DATA_BLOCK "dbdane"   // DB2
{ S7_Optimized_Access := 'FALSE' }
VERSION : 0.1
// stored: AutoNumber true, DBAccessibleFromOPCUA true, IsOnlyStoredInLoadMemory false, IsWriteProtectedInAS false
   VAR RETAIN
      TMR_ON_K3 : Time := T#10s;   // Czas histerezy na dołączenie dodatkowej 3 / Wartość timera na dołączenie drugiej dodatkowej
      amplituda : Real := 95.0;   // Wiekośc zadana amplituda sygnału
      TMR_OFF_K3 : Time := T#10s;   // Czas na odłączenie dodatkowej 3 / Wartość timera na odłączenie drugiej dodatkowej
      Manual_SV : Real;   // Wartość setpint zadana manualnie
      MV : Real;   // Wartość procentowa wyjącia regulatora PID [%]
      PV : Real;   // Wartość liczbowa sygnału analogowego cisnienia tłocznym / Wartość liczbowa sygnału analogowego AI0 bar ciśnienie tłoczenia t
      tuning : Bool;
      zewnetrzne : Bool;
      dzialanie : Bool;
      Setpoint_SV : Real;   // Ciśnienie zadane do regulatora / Wartość zadanego ciśnienia do PID
      WYL : Bool;
      zerowanie : Bool;
      z_obiektu_analog : Word;
      do_obiektu_analog : Word;
      do_obiektu_pwm : Bool;
      PV_PER_B6 : Word;   // Ciśnienie tłoczny miasto (4-20mA) / Ciśnieie Tłoczenia Tłoczny sygnał z wejścia analogowego AI0 bar (4-20mA)
      OUT_PER : Word;   // Sygnał wyjściowy Hz postać procesowa / Sygnał wyjściowy Hz postać analogowa 0-20mA
      TMR_ON_K1 : Time;   // Wartość timera na dołączenie
      TMR_ON_K2 : Time;   // Wartość timera na dołączenie
      TMR_OFF_K1 : Time;   // Wartość timera na odłączenie
      TMR_OFF_K2 : Time;   // Wartość timera na odłączenie
      TMR_Hz : Time;   // Wartość timera na oczykiwanie 50Hz
      HMI : Struct
         PhysicalUnit : String[5] := '1/min';
         Output_PWM_USInt : USInt;
         ManualEnable_edge : Bool;
         ManualMode_visible : Bool;
         "sPid_Cmpt.b_Input_PER_On" : Bool;
         ErrorBits_Int : Int;
         ErrorAck_Int : Int;
         Warning_Int : Int;
         ErrorAck_Int_edge : Bool;
         ErrorAck : Bool;
         Acknowledge_visible : Bool;
         "sPid_Cmpt.r_Pv_Norm_OUT_2" : Real;   // Max wartośc procesowa przekazana z HMI
      END_STRUCT;
      OUT_PURE_Real : Real;   // Sygnał Hz w po scalowaniu do Hz
      Edge_1Hz_P1 : Bool;   // Pamięć zbocza naraztającego dla licznika pracy / Pamięć zbocza naraztającego dla licznika pracy pompy
      Edge_1Hz_P2 : Bool;   // Pamięć zbocza naraztającego dla licznika pracy / Pamięć zbocza naraztającego dla licznika pracy pompy
      Edge_1Hz_P3 : Bool;   // Pamięć zbocza naraztającego dla licznika pracy / Pamięć zbocza naraztającego dla licznika pracy pompy
      Edge_1Hz_P4 : Bool;   // Pamięć zbocza naraztającego dla licznika pracy pompy
      "PID_Compact_1_sPid_Cmpt.r_Lmn_Hlm" : Real;
      "PID_Compact_1sPid_Cmpt.r_Pv_Norm_OUT_2" : Real;
      PID_Compact_1_ManualEnable : Bool;
      PID_Compact_1_ManualValue { ExternalWritable := 'False'} : Real;
      "PID_Compact_1_sPid_Cmpt.r_Lmn_Llm" : Real;
      "PID_Compact_1_sPid_Cmpt.r_Lmn_Pwm_PBTm" : Real;
      "PID_Compact_1_sPid_Cmpt.r_Lmn_Pwm_PPTm" : Real;
      "PID_Compact_1_sPid_Cmpt.r_Pv_HWrn" : Real;   // Nastawa progu ostrzerzenia PV wysoki
      "PID_Compact_1_sPid_Cmpt.r_Pv_LWrn" : Real;   // Nastawa progu ostrzerzenia PV niski
      "PID_Compact_1_sPid_Cmpt.r_Pv_Norm_IN_1" : Real;
      "PID_Compact_1_sPid_Cmpt.r_Pv_Norm_IN_2" : Real;
      "PID_Compact_1_sPid_Cmpt.r_Pv_Norm_OUT_1" : Real;
      "PID_Compact_1_sPid_Cmpt.r_Sp_Hlm" : Real;
      "PID_Compact_1_sPid_Cmpt.r_Sp_Llm" : Real;
      "PID_Compact_1_sPid_Cmpt.r_Pv_Hlm" : Real;
      "PID_Compact_1_sPid_Cmpt.r_Pv_Llm" : Real;
      Setpoint_bar_automat : Real;   // Zadana wartość ciśnienia w trybie automat (sterownik pobiera określoną wartośc zadaną w zależności od kierunku pompowania) / Ciśnienie w magistrali (bobrane ze sterownika Zasuwy) skalowany
      PV_PER_B8 : Word;   // Ciśnienie ssanie suchobieg (4-20mA) / Ciśnienie po stronie ssącej pomp (sychobieg)
      MV_Real_b : Word;
      actPrzepływQ1_Real : Real;   // przepływ pompownia / Aktualny przepływ POMPOWNIA
      actPrzepływQ2_Real : Real;   // Zadane Hz pompomieszadło Word / Aktualny przepływ EC STUDNIA POMIAROWA
      Switch_model_control_Tanks : Word;   // Sygnał sterowania zbiornikami -strategia
      Z11_Status : Word;
      Z12_Status : Word;
      Temp_SV : Word;   // Tymczasowa zadana wartość Hz
      Switch_model_control_P1P4 : Word;   // Sygnały sterowania strategią pompownia - 0= wyłaczone, 1=dosilanie, 2=przetłaczanie,3=automat, 4=ręczne / Model sterowania pompownią (1-dobowe , 2-tygodniowe , 3-Sterowanie standard
      tmp_Hz_ModeAlarm : Real;   // Przechwycone Hz podczas wystąpienia alarmu od max ciśnienie, prąd / Przechwycone Hz podczas wytąpienia alarmu od max ciśnienie, prąd
      actPrzeoływQ1 { ExternalVisible := 'False'} : Int;   // Zmienna aktualny przepływ pompowia / aktualny przepływ Studnia pomiarowa EC Moszczenica
      actPrzepływQ1_IA : Int := 0;   // Zmienna po konwersji do Integer / aktualny przepływ z wejcia analgowego Pompownia jeśli (-) to przepływ wsteczny
      Act_Value_B5_magistrala_bar : Real;   // Zmienna aktualnej wartości ciśnienia magistrala z PLC Zasuwy / Zmienna aktualnej wartości ciśnieniea wspólna Modbus i 4-20mA
      actHz_QW64 : Real := 0.0;   // Zmienna Hz pobrane z wyjacia analogowego / Zmienna aktualnej wartości ciśnieniea wspólna Modbus i 4-20mA
      actPrzepływQ1_IA_real : Real;   // aktualny przepływ Q1 pompownia z wyjścia analogowego / Śerdnia wartość ciśnienie B5 B9
      PV_PER_B7 : Word;   // Ciśnienie tłoczny pompownia(4-20mA) / Ciśnieie Tłoczenia Pompy sygnał z wejścia analogowego AI0 bar (4-20mA)
      act_Value_B6 : Real;   // Ciśnienie tłoczny miasto (Real) / Zmienna aktualnej wartości ciśnieniea B6 po skalowaniau z wejścia (Ciśnieie Tłoczenia Miasto)
      act_Value_B7 : Real;   // Ciśnienie tłoczny pompownia (Real) / Zmienna aktualnej wartości ciśnieniea B7 po skalowaniau z wejścia (Ciśnienie pomp )
      act_Value_B8 : Real;   // Zmienna aktualnej wartości ciśnieniea B5 po skalowaniau z wejścia (Ciśnieie dosilania B5 ) / Ciśnienie ssania (Real)
      tmpdata_MV_PER : Word;   // Tymczasowa aktualnych Hz na potrzeby SCADA przekaznie między tymczasowym Hz a z regulatora PID
      tmpManualSV : LReal;   // pomocnicza przy konwersji wartość zadana manualnie SV
      ManualSV_Int : Int;   // wartość zadana manualnie SV (Word)
      tmpSV_manual_Hold : Int;   // tymczasowa wartość Hz w postaci procesowej podawana na wyjście w czasie podtrzymywania pompy wiodącej po odłaczeniu dodatkowej / tymczasowa wartość Hz w postaci procesowej podawana na wyjście w czasie podtrzymywania dmuchawy wiodącej po odłaczeniu dodatkowej
      tmp_TR_ON_K1_1 : Int := 300;   // Zmienna czasu na dołączenie dodatkowej 1 pobierana przez algorytm PLC
      tmp_TR_ON_K2_1 : Int := 60;   // Zmienna czasu na dołączenie dodatkowej 2 pobierana przez algorytm PLC
      tmp_TR_OFF_K1_1 : Int := 5;   // Zmienna czasu na odołączenie dodatkowej 1 pobierana przez algorytm PLC
      tmp_TR_OFF_K2_1 : Int := 3;   // Zmienna czasu na odołączenie dodatkowej 2 pobierana przez algorytm PLC
      tmp_TR_50Hz_1 : Int := 15;   // Zmienna oczekiwania na 50Hz pobierana przez algorytm PLC
      tmp_TR_ON_K1_2 : Int := 30;   // Zmienna czasu na dołączenie dodatkowej 1 pobierana przez algorytm PLC
      tmp_TR_ON_K2_2 : Int := 30;   // Zmienna czasu na dołączenie dodatkowej 2 pobierana przez algorytm PLC
      tmp_TR_OFF_K1_2 : Int := 5;   // Zmienna czasu na odołączenie dodatkowej 1 pobierana przez algorytm PLC
      tmp_TR_OFF_K2_2 : Int := 5;   // Zmienna czasu na odołączenie dodatkowej 2 pobierana przez algorytm PLC
      tmp_TR_50Hz_2 : Int := 30;   // Zmienna oczekiwania na 50Hz pobierana przez algorytm PLC
      tmp_TR_ON_K1_3 : Int := 5;   // Zmienna czasu na dołączenie dodatkowej 1 pobierana przez algorytm PLC
      tmp_TR_ON_K2_3 : Int := 15;   // Zmienna czasu na dołączenie dodatkowej 2 pobierana przez algorytm PLC
      tmp_TR_OFF_K1_3 : Int := 2;   // Zmienna czasu na odołączenie dodatkowej 1 pobierana przez algorytm PLC
      tmp_TR_OFF_K2_3 : Int := 2;   // Zmienna czasu na odołączenie dodatkowej 2 pobierana przez algorytm PLC
      tmp_TR_50Hz_3 : Int := 5;   // Zmienna oczekiwania na 50Hz pobierana przez algorytm PLC
      tmpSV_spadekBar : Int;   // Hz tymczasowe dla spatku bar Max po odłączeniu dodatkowej / Hz tymczasowe dla opadającego ciśnienia z Max po odłączeniu dodatkowej
      Alarm_Max_bar : Real;   // Alarmowa wartość bar natychmiastowe wyłączenie układu / Alarmowa wartość tlenu natychmiastowe wyłączenie układu
      tmpSV_spadek : Int := 15000;   // pomocnicza Hz tymczasowe dla opadającego ciśnienie z Max / pomocnicza Hz tymczasowe dla opadającego ciśnienia z Max
      addressModbus_Fal : Byte;   // adres modbas urządzenia falownik
      addressModbus_Q1_MPP04 : Byte;   // adres modbas urządzenia przepłuwomierz Q1
      addressModbus_Q2_MPP04 : Byte;   // adres modbas urządzenia przepływomierz Q2
      addressModbus_SlaveID : Byte;   // adres modbas ID slave
      Wielkość_przeływu_Q1 : Real;
      Licznik_objętość_VF_Q1 : Real;
      Licznik_objętość_VR_Q1 : Real;
      Licznik_różnicowy_VD_Q1 : Real;
      Stan_licz_bjętości_GF_Q1 : Real;
      Stan_licz_rózicowego_obj_GD_Q1 : Real;
      _Stan_urządzenia_Q1 : Int;
      Wielkość_przeływu_Q2 : Real;
      Licznik_objętość_VF_Q2 : Real;
      Licznik_objętość_VR_Q2 : Real;
      Licznik_różnicowy_VD_Q2 : Real;
      Stan_licz_bjętości_GF_Q2 : Real;
      Stan_licz_rózicowego_obj_GD_Q2 : Real;
      _Stan_urządzenia_Q2 : Int;
      PV_analaog_B6 : Int;   // wartość analogowa z wejścia AI
      PV_analaog_B7 : Int := 0;   // wartość analogowa z wejścia AI
      PV_analaog_B8 : Int := 0;   // wartość analogowa z wejścia AI
   END_VAR
BEGIN
END_DATA_BLOCK

DATA_BLOCK "dbtags_Sterowanie"   // DB1
{ S7_Optimized_Access := 'FALSE' }
VERSION : 0.1
// stored: AutoNumber false, DBAccessibleFromOPCUA true, IsOnlyStoredInLoadMemory false, IsWriteProtectedInAS false
   VAR RETAIN
      PID_Compact : Struct
         Setpoint : Real := 1.5;
         Input : Real;
         Input_PER : Int;
         Disturbance : Real;
         ManualEnable : Bool;
         ManualValue : Real;
         ErrorAck : Bool;
         Reset : Bool;
         ModeActivate : Bool;
         Mode : Int := 3;
         ScaledInput : Real;
         Output : Real;
         Output_PER : Int;
         Output_PWM : Bool;
         SetpointLimit_H : Bool;
         SetpointLimit_L : Bool;
         InputWarning_H : Bool;
         InputWarning_L : Bool;
         State : Int;
         Error : Bool;
         ErrorBits : DWord;
      END_STRUCT;
      Tuning : Struct
         Mode : Int := 1;
         Mode_visible : Bool;
         SUT_visible : Bool;
         TIR_visible : Bool;
         last_state : Int;
      END_STRUCT;
      HMI : Struct
         PhysicalUnit : String[5] := '1/min';
         Output_PWM_USInt : USInt;
         "position reached" : Bool;
         ManualMode_visible : Bool;
         Setpoint_limited : Bool;
         ErrorBits_Int : Int;
         ErrorAck_Int : Int;
         Warning_Int : Int;
         ErrorAck_Int_edge : Bool;   // pamięć zbocza reset PID po error
         ErrorAck : Bool;   // reset błędu PID
         Acknowledge_visible : Bool;
      END_STRUCT;
      Speed : Struct
         encoder : Real;
         rpm : Real;
      END_STRUCT;
      SetupControlPompownia : Struct
         SV : Real := 2.0;
         r_Pv_Norm_OUT_2 : Real := 10.0;   // Zakres górny wejścia In_PER_PID
         r_Pv_Norm_OUT_1 : Real := 0.0;   // Zakres dolny wejścia In_PER_PID
         r_Lmn_Hlm : Real := 100.0;   // Ograniczenie górne wartości procesowej [%] MV
         r_Lmn_Llm : Real := 0.0;   // Ograniczenie dolne wartości procesowej [%] MV
         r_Sp_Hlm : Real := 10.0;   // Ograniczenie H zakresu zadawania wartości ciśnienie SV
         r_Sp_Llm : Real := 0.0;   // Ograniczenie L zakresu zadawania wartości ciśnienia SV
         r_Pv_HWrn : Real;   // Ostrzeżenie wysoki dla PV
         r_Pv_LWrn : Real;   // Ostrzeżenie niski dla PV
         r_Pv_Hlm : Real := 16.0;   // Przetwornik Limit górny
         r_Pv_Llm : Real := 0.0;   // Przetwornik Limit dlolny
         Time_ONK1 : Int := 20;
         Time_ONK2 : Int := 60;
         Time_OFFK1 : Int := 15;
         Time_OFFK2 : Int := 5;
         TimeHz : Int := 10;
         NO4_Cureent : Real;   // Aktualna zawartość amoniaku
         CureentValue_O2_1 : Real;   // Przyrost ciśnienia 1
         CureentValue_O2_2 : Real;   // Przyrost ciścienia 2
         Data_sek1 : Int;   // Licznik sekund dla pomiaru nr1 funkcji Calculation_of_the_increment
         Data_sek2 : Int;   // Licznik sekund dla pomiaru nr2 funkcji Calculation_of_the_increment
         Static_1 : Word;
         Z11_Status : Word;   // Status napędu copia z SCADA
         Z12_Status : Word;   // Status napędu copia z SCADA
         Static_2 : Real;
         Switch_Aut_Rem_Pompy : Bool;   // Bit przełacznika trybu pracy pomp
         tagsdbSwitch_ModelSterowania : Word;   // Wybur model sterowania0- wyłączone, 1- Dosilanie, 2- Przetłączanie, 3- Automat, 4- Ręczne
         barMax_Manual_Hz : Real := 5.0;   // Instancja wartości zadawanej w trybie manual do regulatora PID gdy ciśnienie w rurociągu max
         CurrentMax_Manual_Hz : Real := 5.0;   // Instancja wartości zadawanej w trybie manual do regulatora PID gdy przeciążony falownik
         Statut_Motor : Byte;   // Byte stanu gotowości pomp
         Mem_Res_setCMD_MC_P1 : Bool;   // Znacznik 50 Hz podtrzymanie przełączenia na sieć
         Mem_Res_setCMD_MC_P2 : Bool;   // Znacznik 50 Hz podtrzymanie przełączenia na sieć
         Mem_Res_setCMD_MC_P3 : Bool;   // Znacznik 50 Hz podtrzymanie przełączenia na sieć
         Switch_In_Analog_Mudbas : Bool;   // Bit przełączeania pomiędzy sygnałem bar z wej analog / Modbus
         PV_HWrn_correction : Real;   // Wspóczninik służący wprowadzeniu korekty ostrzeżenia przekroczenia wartości zadanej ciśnienie
         PV_LWrn_correction : Real;   // Wspóczninik służący wprowadzeniu korekty ostrzeżenia zbyt niskia wartości ciśnieniea w stosunku do zadanej
         TimerSet_O2_Up : IEC_TIMER;   // Czas opóżninia podniesienia zadanej wartości ciśnienia
         TimerSet_O2_Down : IEC_TIMER;   // Czas opóżninia obniżenia zadanej wartości ciśnienia
         Pv_Llm_B8 : Real := -1.0;   // Limit dolny przetwornika ciśnienie B8
         Pv_Hlm_B8 : Real := 2.0;   // Limit górny przetwornika ciśnienia B8
         set_a : Int;
         set_b : Int := 0;
         Setpoint_Inverter_Pompy { ExternalAccessible := 'False'; ExternalVisible := 'False'; ExternalWritable := 'False'} : Real;   // Wartość zadana Hz odczytane z Modbus
         Frequency_inverter_Pompy { ExternalAccessible := 'False'; ExternalVisible := 'False'; ExternalWritable := 'False'} : Real;   // Aktualne Hz silniku odczytane z Modbus
         MotorCurrent_Inverter_Pompy { ExternalAccessible := 'False'; ExternalVisible := 'False'; ExternalWritable := 'False'} : Real;   // Prąd na silniku zasilanym z falownika odczytane z Modbus
         NormalCurrent_InverterPompy { ExternalAccessible := 'False'; ExternalVisible := 'False'; ExternalWritable := 'False'} : Real;   // Prąd nominalny falownika odczytane z Modbus
         MaxCurrent_Inverter_Pompy { ExternalAccessible := 'False'; ExternalVisible := 'False'; ExternalWritable := 'False'} : Real;   // Prad Max krótkotrwały odczytane z Modbus
         OverTemp_InverterPompy { ExternalAccessible := 'False'; ExternalVisible := 'False'; ExternalWritable := 'False'} : Word;
         OverVolta_InverterPompy { ExternalAccessible := 'False'; ExternalVisible := 'False'; ExternalWritable := 'False'} : Word;
         PIF_Reset : IEC_TIMER;   // impuls resetu regulatora PID 1
         mbAdresMPP04_Q1 : Word := 6;   // Adres modbus przepływomierz pompownia
         mbAdresPompy : Word := 26;   // Adres modbus falownik
         mbAdresMPP04_Q2 : Word;   // Adres modbus przepływomierz magistrala - w Stacji Zasuw
         mbAdres_IDslave : Word := 2;   // Adres modbus MT101
         SubPV_K1 : Real := 0.6;   // Wspólczynnik pomniejszenia wyliczanego ciśnienia napotrzeby wyłączenia dodatowej pompy
         SubPV_K2 : Real := 0.45;   // Wspólczynnik pomniejszenia wyliczanego ciśnieia napotrzeby wyłączenia dodatowej pompy
         Setpoint_Inverter_a { ExternalAccessible := 'False'; ExternalVisible := 'False'; ExternalWritable := 'False'} : Real;   // Wartość zadana Hz odczytane z Modbus
         Frequency_inverter_a { ExternalAccessible := 'False'; ExternalVisible := 'False'; ExternalWritable := 'False'} : Real;   // Aktualne Hz silniku odczytane z Modbus
         MotorCurrent_Inverter_a { ExternalAccessible := 'False'; ExternalVisible := 'False'; ExternalWritable := 'False'} : Real;   // Prąd na silniku zasilanym z falownika odczytane z Modbus
         NormalCurrent_Inverter_a { ExternalAccessible := 'False'; ExternalVisible := 'False'; ExternalWritable := 'False'} : Real;   // Prąd nominalny falownika odczytane z Modbus
         MaxCurrent_Inverter_a { ExternalAccessible := 'False'; ExternalVisible := 'False'; ExternalWritable := 'False'} : Real;   // Prad Max krótkotrwały odczytane z Modbus
         OverTemp_InverterPomp { ExternalAccessible := 'False'; ExternalVisible := 'False'; ExternalWritable := 'False'} : Word;
         OverVolta_InverterPomp { ExternalAccessible := 'False'; ExternalVisible := 'False'; ExternalWritable := 'False'} : Word;
         set_barDN500_B5 { ExternalAccessible := 'False'; ExternalVisible := 'False'; ExternalWritable := 'False'} : Real;   // Zadane ciśnienie dosilanie DN500 na czujniku B5
         set_barDN225_B6 { ExternalAccessible := 'False'; ExternalVisible := 'False'; ExternalWritable := 'False'} : Real;   // Zadane ciśnienie przetłacania DN225 na czujniku B6
         MotorCurrent_Inverter_b { ExternalAccessible := 'False'; ExternalVisible := 'False'; ExternalWritable := 'False'} : Real;   // Prąd na silniku zasilanym z falownika odczytane z Modbus
         NormalCurrent_Inverter_b { ExternalAccessible := 'False'; ExternalVisible := 'False'; ExternalWritable := 'False'} : Real;   // Prąd nominalny falownika odczytane z Modbus
         MaxCurrent_Inverter_b { ExternalAccessible := 'False'; ExternalVisible := 'False'; ExternalWritable := 'False'} : Real;   // Prad Max krótkotrwały odczytane z Modbus
         OverTemp_Inverter_b { ExternalAccessible := 'False'; ExternalVisible := 'False'; ExternalWritable := 'False'} : Word;
         OverVolta_Inverter_b { ExternalAccessible := 'False'; ExternalVisible := 'False'; ExternalWritable := 'False'} : Word;
         actOverCurrent_set : Real;   // Zakres ograniczenia prądowego.
         actOverCurrent_set_a : Real := 0.0;   // Zakres ograniczenia prądowego.
         actOverCurrent_set_b : Real := 0.0;   // Zakres ograniczenia prądowego.
         AnalogFrequency_inverter_a { ExternalAccessible := 'False'; ExternalVisible := 'False'; ExternalWritable := 'False'} : Real;   // Aktualne Hz silniku odczytane z Analog
         AnalogFrequency_inverter_b { ExternalAccessible := 'False'; ExternalVisible := 'False'; ExternalWritable := 'False'} : Real := 0.0;   // Aktualne Hz silniku odczytane z Analog
         MaxHour_InverterBlowerWork : Word := 43200;   // Maksymalny czas pracy pracy ciągłej na falowniku dla kompresorów 43200sek = 12h
         TimerSet_Hz_Up_a : IEC_TIMER;
         TimerSet_Hz_Down_a : IEC_TIMER;
         TimerSet_Hz_Up_b : IEC_TIMER;
         TimerSet_Hz_Down_b : IEC_TIMER;
         TimerGen_Hz_Up_a : IEC_TIMER;
         TimerGen_Hz_Down_a : IEC_TIMER;
         TimerGen_Hz_Up_b : IEC_TIMER;
         TimerGen_Hz_Down_b : IEC_TIMER;
         Mem_Res_setCMD_MC_P4 : Bool;   // Znacznik 50 Hz podtrzymanie przełączenia na sieć
         "MPP04_1Master.mode" : Byte := 0;
         "MPP04_2Master.mode" : Byte := 0;
         "Fal_2Master.mode_1" : Byte := 0;
         "Slave_2Master.mode_2" : Byte := 2;
      END_STRUCT;
      "Paramaetry _Zbiorniki" : Struct   // parametry sterowania
         set_poziom_napełniania : Real := 550.0;   // wartość zadana poziomu napełniania
         set_poziom_opróżniania : Real := 30.0;   // wartość zadana poziomu opróżniania
         set_bity_sterowania_napęami_1 : Word;   // bity sterowania napędami
         set_bity_sterowania_napęami_2 : Word;   // bity sterowania napędami
         set_bity_tryb_napędów_1 : Word;   // bity sterowania przełączaniem trybów pracy
         set_bity_tryb_napędów_2 : Word;   // bity sterowania przełączaniem trybów pracy
         rez_alarm_napędów : Word;   // bity kasowania alarmów napędów
         set_strategia_sterowania : Word;   // Sygnały sterowania strategią pompownia - 0= wyłaczone, 1=dosilanie, 2=przetłaczanie,3=automat, 4=ręczne
         set_sterowanie_cyklem : Word;   // Sygnały sterowania cyklem zbiorniki 0-wyłączone, 1=dobowy, 2=tygodniowy, 3=ręczne
         set_położenie_Z10 : Word;   // zadane położenie procentowe Z10
      END_STRUCT;
      Zbiorniki_Godziny : Struct   // godziny cykli pracy
         start_napełnianie : DTL := DTL#1970-01-01-23:55:00;
         Stop_napełnianie : DTL := DTL#1970-01-01-16:00:00;
         Start_przetłaczanie_1 : DTL := DTL#1970-01-01-18:00:00;
         Stop_przetłaczanie_1 : DTL := DTL#1970-01-01-23:55:00;
         Start_dosilanie_1 : DTL := DTL#1970-01-01-18:00:00;
         Stop_dosilanie_1 : DTL := DTL#1970-01-01-23:55:00;
      END_STRUCT;
   END_VAR
BEGIN
   SetupControlPompownia.PIF_Reset.PT := T#500ms;
   SetupControlPompownia.TimerSet_Hz_Up_a.PT := T#2M;
   SetupControlPompownia.TimerSet_Hz_Down_a.PT := T#2M;
   SetupControlPompownia.TimerSet_Hz_Up_b.PT := T#2M;
   SetupControlPompownia.TimerSet_Hz_Down_b.PT := T#2M;
   SetupControlPompownia.TimerGen_Hz_Up_a.PT := T#100ms;
   SetupControlPompownia.TimerGen_Hz_Down_a.PT := T#100ms;
   SetupControlPompownia.TimerGen_Hz_Up_b.PT := T#100ms;
   SetupControlPompownia.TimerGen_Hz_Down_b.PT := T#100ms;
END_DATA_BLOCK

DATA_BLOCK "dbMasterData"   // DB35
{ S7_Optimized_Access := 'FALSE' }
VERSION : 0.1
// stored: AutoNumber false, DBAccessibleFromOPCUA true, IsOnlyStoredInLoadMemory false, IsWriteProtectedInAS false
   VAR
      data5_Wielkość_przeływu_Adres_0 { S7_SetPoint := 'True'} : "typeDataMPP04_Int";   // wielkość przepływu / Wartość aktualnego przepływu
      data5_Licznik_objętość_VF_Adres_2 : "typeDataMPP04_Int";   // licznik objętości VF / Stan licznika objętości dla przepływu w przód VF
      data5_Licznik_objętość_VR_Adres_4 { S7_SetPoint := 'True'} : "typeDataMPP04_Int";   // licznik objętości VR / Stan licznika objętości dla przepływu w tył VR
      data5_Licznik_różnicowy_VD_Adres_6 { S7_SetPoint := 'True'} : "typeDataMPP04_Int";   // licznik różnicy / Stan bieżącego różnicowego licznika objętości VD
      data5_Stan_licz_bjętości_GF_Adres_8 { S7_SetPoint := 'True'} : "typeDataMPP04_Int";   // licznik objetosci GF / Stan głównego licznika objętości dla przepływu w przód GF
      data5_Stan_licz_bjętości_GR_Adres_10 { S7_SetPoint := 'True'} : "typeDataMPP04_Int";   // licznik objetości GR / Sta ngłownego licznika objętości dla przepływu w tył GR
      data5_Stan_licz_rózicowego_obj_GD_Adres_12 { S7_SetPoint := 'True'} : "typeDataMPP04_Int";   // licznik róznicowy / Stan głownego licznika różnicowego GD
      data5_Stan_urządzenia_1000 { S7_SetPoint := 'True'} : "typeDataInverter_Word";   // stan urządzenia / 8-przekrodzony zakres pracy przetwornika, 20-otwarty obwód cewki, 21zwarcie w obwodzie cewki, 26-brak cieczy w czujniku
      data6_Wielkość_przeływu_Adres_0 { S7_SetPoint := 'True'} : "typeDataMPP04_Int";   // wielkość przepływu / Wartość aktualnego przepływu
      data6_Licznik_objętość_VF_Adres_2 { S7_SetPoint := 'True'} : "typeDataMPP04_Int";   // licznik objętości VF / Stan licznika objętości dla przepływu w przód VF
      data6_Licznik_objętość_VR_Adres_4 { S7_SetPoint := 'True'} : "typeDataMPP04_Int";   // licznik objętości VR / Stan licznika objętości dla przepływu w tył VR
      data6_Licznik_różnicowy_VD_Adres_6 { S7_SetPoint := 'True'} : "typeDataMPP04_Int";   // licznik różnicy / Stan bieżącego różnicowego licznika objętości VD
      data6_Stan_licz_bjętości_GF_Adres_8 { S7_SetPoint := 'True'} : "typeDataMPP04_Int";   // licznik objetosci GF / Stan głównego licznika objętości dla przepływu w przód GF
      data6_Stan_licz_bjętości_GR_Adres_10 { S7_SetPoint := 'True'} : "typeDataMPP04_Int";   // licznik objetości GR / Sta ngłownego licznika objętości dla przepływu w tył GR
      data6_Stan_licz_rózicowego_obj_GD_Adres_12 { S7_SetPoint := 'True'} : "typeDataMPP04_Int";   // licznik róznicowy / Stan głownego licznika różnicowego GD
      data6_Stan_urządzenia_1000 { S7_SetPoint := 'True'} : "typeDataInverter_Word";   // stan urządzenia / 8-przekrodzony zakres pracy przetwornika, 20-otwarty obwód cewki, 21zwarcie w obwodzie cewki, 26-brak cieczy w czujniku
      data26_Inver_Control_word_416000_Fal { S7_SetPoint := 'True'} : "typeDataInverter_Word";   // Sowo komtrolneCTW falownika [Uint16, index 0]
      data26_Inver_setpoint_ref_416020_Fal { S7_SetPoint := 'True'} : "typeDataInverter_Word";   // Słowo wartość zadana Hz [Int16, index -1]
      data26_Inver_Status_word_416030_Fal { S7_SetPoint := 'True'} : "typeDataInverter_Word";   // Słowo statusu STW falownika [Uint16, index 0]
      data26_Inver_Frequency_416130_Fal { S7_SetPoint := 'True'} : "typeDataInverter_Word";   // Słowo częstotliwość na wyjściu [Uint16, index -1]
      data26_Inver_MotorCurrent_416140_Fal { S7_SetPoint := 'True'} : "typeDataInverter_Word";   // Słowo częstotliwość na wyjściu [Uint16, index -2]
      data26_Inver_DC_Voltage_416300_Fal { S7_SetPoint := 'True'} : "typeDataInverter_Word";   // Słowo napięcia DC na szynie [Uint16, index 0]
      data26_Inver_Temp_416340_Fal { S7_SetPoint := 'True'} : "typeDataInverter_Word";   // Słowo temperatura invertera [Uint8, index 0]
      data26_Inver_NomCurrent_416360_Fal { S7_SetPoint := 'True'} : "typeDataInverter_Word";   // Słowo nominalna wartośc prądu falonika[Uint16, index -2]
      data26_Inver_MaxCurrent_416370_Fal { S7_SetPoint := 'True'} : "typeDataInverter_Word";   // Słowo max prąd falownika [Uint16, index -2]
      data26_Inver_InDigit_416600_Fal { S7_SetPoint := 'True'} : "typeDataInverter_Word";   // Słowo mampa wejść 18,19,27,33 [Uint16, index -0]
      data26_Inver_HourWork_415010_Fal { S7_SetPoint := 'True'} : "typeDataInverter_DWord";   // Podwójne słowo czasu pracy falownika [Int32, index -0]
      data26_Inver_OverTemp_415040_Fal { S7_SetPoint := 'True'} : "typeDataInverter_Word";   // Sowo statusu przekroczenie temperatury[Uint16, index 0]
      data26_Inver_OverVolts_415050_Fal { S7_SetPoint := 'True'} : "typeDataInverter_Word";   // Sowo statusu przekroczenie napięcia[Uint16, index 0]
      data_RTU_value_0 { S7_SetPoint := 'True'} : "typeDataMPP04_real";   // Wartość 0.0 pomocnicza wyświetlana podczas błędu pomiaru
   END_VAR
BEGIN
   data_RTU_value_0.data[0] := 0.0;
END_DATA_BLOCK

DATA_BLOCK "dbModbusRTU_Reg"   // DB37
TITLE = Modbus RTU Data
{ S7_Optimized_Access := 'FALSE' }
AUTHOR : RTecmer
VERSION : 0.1
// Dane pomiarowe przekazane z bloku danych master modbus RTU
// stored: AutoNumber true, DBAccessibleFromOPCUA true, IsOnlyStoredInLoadMemory false, IsWriteProtectedInAS false
   VAR
      received_5_Wielkość_przeływu_Adres_0 { S7_SetPoint := 'True'} : "typeDataMPP04_Int";   // wielkość przepływu
      received_5_Licznik_objętość_VF_Adres_2 { S7_SetPoint := 'True'} : "typeDataMPP04_Int";   // licznik objętości VF
      received_5_Licznik_objętość_VR_Adres_4 { S7_SetPoint := 'True'} : "typeDataMPP04_Int";   // licznik objętości VR
      received_5_Licznik_różnicowy_VD_Adres_6 { S7_SetPoint := 'True'} : "typeDataMPP04_Int";   // licznik różnicy
      receive_5_Stan_licz_bjętości_GF_Adres_8 { S7_SetPoint := 'True'} : "typeDataMPP04_Int";   // licznik objetosci GF
      received_5_Stan_licz_bjętości_GR_Adres_10 { S7_SetPoint := 'True'} : "typeDataMPP04_Int";   // licznik objetości GR
      received_5_Stan_licz_rózicowego_obj_GD_Adres_12 { S7_SetPoint := 'True'} : "typeDataMPP04_Int";   // licznik róznicowy
      received_5_Stan_urządzenia_1000 { S7_SetPoint := 'True'} : "typeDataInverter_Word";   // stan urządzenia
      received_6_Wielkość_przeływu_Adres_0 { S7_SetPoint := 'True'} : "typeDataMPP04_Int";   // wielkość przepływu
      received_6_Licznik_objętość_VF_Adres_2 { S7_SetPoint := 'True'} : "typeDataMPP04_Int";   // licznik objętości VF
      received_6_Licznik_objętość_VR_Adres_4 { S7_SetPoint := 'True'} : "typeDataMPP04_Int";   // licznik objętości VR
      received_6_Licznik_różnicowy_VD_Adres_6 { S7_SetPoint := 'True'} : "typeDataMPP04_Int";   // licznik różnicy
      receive_6_Stan_licz_bjętości_GF_Adres_8 { S7_SetPoint := 'True'} : "typeDataMPP04_Int";   // licznik objetosci GF
      received_6_Stan_licz_bjętości_GR_Adres_10 { S7_SetPoint := 'True'} : "typeDataMPP04_Int";   // licznik objetości GR
      received_6_Stan_licz_rózicowego_obj_GD_Adres_12 { S7_SetPoint := 'True'} : "typeDataMPP04_Int";   // licznik róznicowy
      received_6_Stan_urządzenia_1000 { S7_SetPoint := 'True'} : "typeDataInverter_Word";   // stan urządzenia
      receivede26_Inver_Control_word_416000 { S7_SetPoint := 'True'} : "typeDataInverter_Word";   // Sowo komtrolneCTW falownika [Uint16, index 0]
      received26_Inver_setpoint_ref_416020 { S7_SetPoint := 'True'} : "typeDataInverter_Word";   // Słowo wartość zadana Hz [Int16, index -1]
      received26_Inver_Status_word_416030 { S7_SetPoint := 'True'} : "typeDataInverter_Word";   // Słowo statusu STW falownika [Uint16, index 0]
      received26_Inver_Frequency_416130 { S7_SetPoint := 'True'} : "typeDataInverter_Word";   // Słowo częstotliwość na wyjściu [Uint16, index -1]
      received26_Inver_MotorCurrent_416140 { S7_SetPoint := 'True'} : "typeDataInverter_Word";   // Słowo częstotliwość na wyjściu [Uint16, index -2]
      received26_Inver_DC_Voltage_416300 { S7_SetPoint := 'True'} : "typeDataInverter_Word";   // Słowo napięcia DC na szynie [Uint16, index 0]
      received26_Inver_Temp_416340 { S7_SetPoint := 'True'} : "typeDataInverter_Word";   // Słowo temperatura invertera [Uint8, index 0]
      received26_Inver_NomCurrent_416360 { S7_SetPoint := 'True'} : "typeDataInverter_Word";   // Słowo nominalna wartośc prądu falonika[Uint16, index -2]
      received26_Inver_MaxCurrent_416370 { S7_SetPoint := 'True'} : "typeDataInverter_Word";   // Słowo max prąd falownika [Uint16, index -2]
      received26_Inver_InDigit_416600 { S7_SetPoint := 'True'} : "typeDataInverter_Word";   // Słowo mampa wejść 18,19,27,33 [Uint16, index -0]
      received26_Inver_HourWork_415010 { S7_SetPoint := 'True'} : "typeDataInverter_DWord";   // Podwójne słowo czasu pracy falownika [Int32, index -0]
      received26_Inver_OverTemp_415040 { S7_SetPoint := 'True'} : "typeDataInverter_Word";   // Sowo statusu przekroczenie temperatury[Uint16, index 0]
      received26_Inver_OverVolts_415050 { S7_SetPoint := 'True'} : "typeDataInverter_Word";   // Sowo statusu przekroczenie napięcia[Uint16, index 0]
      "Przepływomierz nr1 pompownia" : Struct
         received_5_przeływu_VF_Adres_0 { S7_SetPoint := 'True'} : Real;
         received_5_objętość_VF_Adres_2 { S7_SetPoint := 'True'} : Real;
         "received_5_objętośc RF_Adres_4" { S7_SetPoint := 'True'} : Real;
         received_5_licznik_różnicowy_VD_Adres_6 { S7_SetPoint := 'True'} : Real;
         received_5_licznik_objętości_GF_Adres_8 { S7_SetPoint := 'True'} : Real;
         received_5_Licznik_objętości_GR_Adres_10 { S7_SetPoint := 'True'} : Real;
         received_5_Licznik_różnicowy_GD_Adres_12 { S7_SetPoint := 'True'} : Real;
         received_5_status_przepływomierza_Adres_1000 { S7_SetPoint := 'True'} : Word;
      END_STRUCT;
      "Przepływomierz nr2 Zasuwy" : Struct
         received_6_przeływu_VF_Adres_0 { S7_SetPoint := 'True'} : Real;
         received_6_objętość_VF_Adres_2 { S7_SetPoint := 'True'} : Real;
         "received_6_objętośc RF_Adres_4" { S7_SetPoint := 'True'} : Real;
         received_6_licznik_różnicowy_VD_Adres_7 { S7_SetPoint := 'True'} : Real;
         received_6_licznik_objętości_GF_Adres_8 { S7_SetPoint := 'True'} : Real;
         received_6_Licznik_objętości_GR_Adres_10 { S7_SetPoint := 'True'} : Real;
         received_6_Licznik_różnicowy_GD_Adres_12 { S7_SetPoint := 'True'} : Real;
         received_6_status_przepływomierza_Adres_1000 { S7_SetPoint := 'True'} : Word;
      END_STRUCT;
   END_VAR
BEGIN
END_DATA_BLOCK

DATA_BLOCK "dbTags_master_Fal_1"   // DB74
{ S7_Optimized_Access := 'FALSE' }
VERSION : 0.1
// stored: AutoNumber true, DBAccessibleFromOPCUA true, IsOnlyStoredInLoadMemory false, IsWriteProtectedInAS false
   VAR
      "step" : USInt := 1;
      edge : Bool := false;
      modbusCommLoad { S7_SetPoint := 'True'} : "typeModbusCommLoad";
      modbusMaster { S7_SetPoint := 'True'} : "typeModbusMaster";
   END_VAR
BEGIN
END_DATA_BLOCK

DATA_BLOCK "dbTags_master_MPP04_1"   // DB38
{ S7_Optimized_Access := 'FALSE' }
VERSION : 0.1
// stored: AutoNumber true, DBAccessibleFromOPCUA true, IsOnlyStoredInLoadMemory false, IsWriteProtectedInAS false
   VAR
      "step" : USInt := 1;
      edge : Bool := false;
      modbusCommLoad { S7_SetPoint := 'True'} : "typeModbusCommLoad";
      modbusMaster { S7_SetPoint := 'True'} : "typeModbusMaster";
   END_VAR
BEGIN
END_DATA_BLOCK

DATA_BLOCK "dbTags_master_MPP04_2"   // DB81
{ S7_Optimized_Access := 'FALSE' }
VERSION : 0.1
// stored: AutoNumber true, DBAccessibleFromOPCUA true, IsOnlyStoredInLoadMemory false, IsWriteProtectedInAS false
   VAR
      "step" : USInt := 1;
      edge : Bool := false;
      modbusCommLoad { S7_SetPoint := 'True'} : "typeModbusCommLoad";
      modbusMaster { S7_SetPoint := 'True'} : "typeModbusMaster";
   END_VAR
BEGIN
END_DATA_BLOCK

DATA_BLOCK "dbTags_master_RTU"   // DB90
TITLE = Master
{ S7_Optimized_Access := 'FALSE' }
AUTHOR : rtecmer
VERSION : 0.1
// Instancja dla funkcji Mdbus RTU komunikacja z masterem MT101
// stored: AutoNumber false, DBAccessibleFromOPCUA true, IsOnlyStoredInLoadMemory false, IsWriteProtectedInAS false
   VAR
      "step" : USInt := 1;
      edge : Bool := false;
      modbusCommLoad { S7_SetPoint := 'True'} : "typeModbusCommLoad";
      modbusMaster { S7_SetPoint := 'True'} : "typeModbusSlave";
   END_VAR
BEGIN
END_DATA_BLOCK

DATA_BLOCK "dbTags_slave_RTU"   // DB79
TITLE = Master
{ S7_Optimized_Access := 'FALSE' }
AUTHOR : rtecmer
VERSION : 0.1
// Instancja dla funkcji Mdbus RTU komunikacja z masterem MT101
// stored: AutoNumber false, DBAccessibleFromOPCUA true, IsOnlyStoredInLoadMemory false, IsWriteProtectedInAS false
   VAR
      "step" : USInt := 1;
      edge : Bool := false;
      modbusCommLoad { S7_SetPoint := 'True'} : "typeModbusCommLoad";
      modbusMaster { S7_SetPoint := 'True'} : "typeModbusSlave";
   END_VAR
BEGIN
END_DATA_BLOCK

DATA_BLOCK "temp_dbHoldRegSlave_to_MT101"   // DB102
{ S7_Optimized_Access := 'FALSE' }
VERSION : 0.1
// stored: AutoNumber false, DBAccessibleFromOPCUA true, IsOnlyStoredInLoadMemory false, IsWriteProtectedInAS false
   VAR
      Status_Sterowanie : Struct
         instPump1 : Int;   // Pompa Status M1
         instPump2 : Int := 0;   // Pompa Status M2
         instPump3 : Int := 0;   // Pompa Status M3
         instPump4 : Int := 0;   // Pompa Status M4
         instvValveZ1 : Int := 0;   // Zasuwa Status Z1
         instvValveZ2 : Int := 0;   // Zasuwa Status Z2
         instvValveZ3 : Int := 0;   // Zasuwa Status Z3
         instvValveZ4 : Int := 0;   // Zasuwa Status Z4
         instvValveZ5 : Int := 0;   // Zasuwa Status Z5
         instvValveZ6 : Int := 0;   // Zasuwa Status Z6
         instvValveZ7 : Int := 0;   // Zasuwa Status Z7
         instvValveZ8 : Int := 0;   // Zasuwa Status Z8
         instvValveZ9 : Int := 0;   // Zasuwa Status Z9
         instvValveZ10 : Int := 0;   // Zasuwa Status Z10
         instvValveZ11 : Int := 0;   // Zasuwa Status Z11
         instvValveZ12 : Int := 0;   // Zasuwa Status Z12
         instControllDrivers_1 : Int := 0;   // Bity sterowania napędami (start, stop, otwórz, zamknij) / Bity sterowania napędami (start, stop, otwórz, zamknij) Pompami M1-M4, Zasuwami Z1, Z2, Z3, Z4
         instControllDrivers_2 : Int := 0;   // Bity przełączenia trybu pracy napędów / Bity sterowania napędami ( otwórz, zamknij, start, stop) Zasuwami Z5, Z6, Z7, Z8, Z9, Z10, Z11, Z12
         instConrol_ManAut_1 : Int := 0;   // Bity przełączenia trybu pracy napędów / Bity przełączenia trybu pracy napędów M1-M4, Zasuwami Z1, Z2, Z3, Z4
         instConrol_ManAut_2 : Int := 0;   // Bity przełączenia trybu pracy napędów / Bity przełączenia trybu pracy napędów Z5, Z6, Z7, Z8, Z9, Z10, Z11, Z12
         instLevelTank1 : Int := 0;   // Poziom zbiornik
         instLevelTank2 : Int := 0;   // Poziom zbiornik
         instLevelTank3 : Int := 0;   // Poziom zbiornik
         instLevelTank4 : Int := 0;   // Poziom zbiornik
         instPosition_Z10 : Int := 0;   // rezerwa / Zadawanie położenia Z10
         instControlClearFault1 : Int := 0;   // Bity kasowania alarmów napędów M1-M4, Z1 - Z12
         instControlSygSter_1 : Int := 0;   // rezerwa / Sygnały sterowania strategią (Bit 53.0 - Wyłączony), (Bit 53.1 - Dosilanie), (Bit 53.2 - Przetłączanie), (Bit 53.3 - Automat), (Bit 53.4 - Ręczne )
         instControlSygSter_2 : Int := 0;   // Sygnały sterowania cyklem (Bit 55.0 - Cykl wyłączony (Bit 55.1 - Cykl dobowy), (Bit 55.2 - Cykl tygodniowy), (Bit 55.3 - Cykl ręczny)
         instCurrent_Inverter : Int := 0;   // Aktualny prądu falownika
         instHz_Inverter : Int := 0;   // Aktualne Hz na falowniku
      END_STRUCT;
      Pomiary : Struct
         instLevelSetfilling : Real;   // Zadany poziom napełniania
         instLevelSetemptying : Real;   // Zadany poziom opróżniania
         instSetbarDN500_B6 : Real;   // Zadany ciśnienie tłóczenia kierunek miasto, Modbus 40035
         instSetbarDN500_B5 : Real;   // Zadana ciśnienie dosilania kierunek dosilanie "0" Modbus 40037
         instSetBarMinB9 : Real;   // Zadawana dolna granica ciśnienia studnia "Granica" Modbus 40039
         instB5bar_act : Real;   // Aktualne ciśnienie zasilania z sieci
         instB6bar_act : Real;   // Aktualne ciśnienie DN225 tłoczny
         instB7bar_act : Real;   // Aktualne ciśnienie DN225 pompy
         instB8bar_act : Real;   // Aktualne ciśnienie ssoncy pomp (zab. Suchobieg)
         instPozitionZ10_act : Real;   // Aktualna pozycja zasuwy Z10
         instFlowDN225_act : Real;   // Przepływ DN225 aktualny MIASTO
         instFlowDN225_sum : Real;   // SUMA przepływu Dolna DN225
         instFlowDN500_act : Real;   // Przepływ DN500 (l/s) aktualny, zasilanie zbiorników, DOSILANIE, Modbus 40055
         instFlowDN500_sum : Real;   // SUMA przepływu Dolna DN500 Modbus 40057
      END_STRUCT;
      Godziny : Struct
         instHourStart_Filling : Int;   // Godzina start napełniania
         instMinutStart_Filling : Int;   // Minuta start napełniania
         instHourStop_Filling : Int;   // Godzina stop napełniania
         instMinutStopt_Filling : Int;   // Minuta stop napełniania
         instHourStart_City : Int;   // Godzina start przetłaczanie miasto DN225
         instMinutStart_City : Int;   // Minuty start przetłaczanie miasto DN225
         instHourStop_City : Int;   // Godzina stop przetłaczanie miasto DN225
         instMinutStopt_City : Int;   // Minuty stop przetłaczanie miasto DN225
         instHourStart_Replen : Int;   // Godzina start przetłaczanie miasto DN225
         instMinutStart_Replen : Int;   // Minuty start przetłaczanie miasto DN225
         instHourStop_Replen : Int;   // Godzina stop przetłaczanie miasto DN225
         instMinutStopt_Replen : Int;   // Minuty stop przetłaczanie miasto DN225
      END_STRUCT;
   END_VAR
BEGIN
END_DATA_BLOCK

DATA_BLOCK "CONFIG_MODBUS_TCP_SERVER"   // DB86
TITLE = CONECT MODBUS TCP SERVER
{ S7_Optimized_Access := 'TRUE' }
AUTHOR : rtecmer
VERSION : 0.1
// stored: AutoNumber true, DBAccessibleFromOPCUA true, IsOnlyStoredInLoadMemory false, IsRetainMemResEnabled false, IsWriteProtectedInAS false, MemoryReserve 100
   VAR
      CONNECT_MODBUS_TCP_Serwer_1 { S7_SetPoint := 'True'} : TCON_IP_v4;
      ERROR_STATUS_SERWER_1 : Word;   // wartość błędu
      ERROR_STATUS_SERWER_2 : Word := 16#0;   // wartość błędu
      ERROR_STATUS_SERWER_3 : Word := 16#0;   // wartość błędu
      ERROR_STATUS_SERWER_4 : Word := 16#0;   // wartość błędu
      "CONFIG SERWER_1" : Struct
         STATUS { S7_SetPoint := 'True'} : Word;   // Status połączenia TCP Modbus
         error : Bool;   // błąd
         dr : Bool;   // dane czytane
         ndr : Bool;   // dane gotowe
      END_STRUCT;
      "CONFIG SERWER_2" : Struct
         STATUS { S7_SetPoint := 'True'} : Word;   // Status połączenia TCP Modbus
         error : Bool;   // błąd
         dr : Bool;   // dane czytane
         ndr : Bool;   // dane gotowe
      END_STRUCT;
      "CONFIG SERWER_3" : Struct
         STATUS { S7_SetPoint := 'True'} : Word;   // Status połączenia TCP Modbus
         error : Bool;   // błąd
         dr : Bool;   // dane czytane
         ndr : Bool;   // dane gotowe
      END_STRUCT;
      "CONFIG SERWER_4" : Struct
         STATUS { S7_SetPoint := 'True'} : Word;   // Status połączenia TCP Modbus
         error : Bool;   // błąd
         dr : Bool;   // dane czytane
         ndr : Bool;   // dane gotowe
      END_STRUCT;
      "CONFIG SERWER_5" : Struct
         STATUS { S7_SetPoint := 'True'} : Word;   // Status połączenia TCP Modbus
         error : Bool;   // błąd
         dr : Bool;   // dane czytane
         ndr : Bool;   // dane gotowe
      END_STRUCT;
      "CONFIG SERWER_6" : Struct
         STATUS { S7_SetPoint := 'True'} : Word;   // Status połączenia TCP Modbus
         error : Bool;   // błąd
         dr : Bool;   // dane czytane
         ndr : Bool;   // dane gotowe
      END_STRUCT;
      "CONFIG SERWER_7" : Struct
         STATUS { S7_SetPoint := 'True'} : Word;   // Status połączenia TCP Modbus
         error : Bool;   // błąd
         dr : Bool;   // dane czytane
         ndr : Bool;   // dane gotowe
      END_STRUCT;
      "CONFIG SERWER_8" : Struct
         STATUS { S7_SetPoint := 'True'} : Word;   // Status połączenia TCP Modbus
         error : Bool;   // błąd
         dr : Bool;   // dane czytane
         ndr : Bool;   // dane gotowe
      END_STRUCT;
      ERROR_STATUS_SERWER_5 : Word := 16#0;   // wartość błędu
      ERROR_STATUS_SERWER_6 : Word := 16#0;   // wartość błędu
      ERROR_STATUS_SERWER_7 : Word := 16#0;   // wartość błędu
      ERROR_STATUS_SERWER_8 : Word := 16#0;   // wartość błędu
   END_VAR
BEGIN
   CONNECT_MODBUS_TCP_Serwer_1.InterfaceId := 64;
   CONNECT_MODBUS_TCP_Serwer_1.ID := 1;
   CONNECT_MODBUS_TCP_Serwer_1.ConnectionType := 11;
   CONNECT_MODBUS_TCP_Serwer_1.LocalPort := 502;
END_DATA_BLOCK

DATA_BLOCK "dbHoldTempMT101"   // DB116
{ S7_Optimized_Access := 'FALSE' }
VERSION : 0.1
// stored: AutoNumber false, DBAccessibleFromOPCUA true, IsOnlyStoredInLoadMemory false, IsWriteProtectedInAS false
   VAR
      Status_Sterowanie : Struct
         instPump1 : Word := 33924;   // Pompa Status M1
         instPump2 : Word := 33924;   // Pompa Status M2
         instPump3 : Word := 33924;   // Pompa Status M3
         instPump4 : Word := 33924;   // Pompa Status M4
         instvValveZ1 : Word := 33924;   // Zasuwa Status Z1
         instvValveZ2 : Word := 33924;   // Zasuwa Status Z2
         instvValveZ3 : Word := 33924;   // Zasuwa Status Z3
         instvValveZ4 : Word := 33924;   // Zasuwa Status Z4
         instvValveZ5 : Word := 33924;   // Zasuwa Status Z5
         instvValveZ6 : Word := 33924;   // Zasuwa Status Z6
         instvValveZ7 : Word := 33924;   // Zasuwa Status Z7
         instvValveZ8 : Word := 33924;   // Zasuwa Status Z8
         instvValveZ9 : Word := 33924;   // Zasuwa Status Z9
         instvValveZ10 : Word := 33924;   // Zasuwa Status Z10
         instvValveZ11 : Word := 33924;   // Zasuwa Status Z11
         instvValveZ12 : Word := 33924;   // Zasuwa Status Z12
         instControllDrivers_1 : Int := 0;   // Bity sterowania napędami (start, stop, otwórz, zamknij) / Bity sterowania napędami (start, stop, otwórz, zamknij) Pompami M1-M4, Zasuwami Z1, Z2, Z3, Z4
         instControllDrivers_2 : Int := 0;   // Bity przełączenia trybu pracy napędów / Bity sterowania napędami ( otwórz, zamknij, start, stop) Zasuwami Z5, Z6, Z7, Z8, Z9, Z10, Z11, Z12
         instConrol_ManAut_1 : Int := 0;   // Bity przełączenia trybu pracy napędów / Bity przełączenia trybu pracy napędów M1-M4, Zasuwami Z1, Z2, Z3, Z4
         instConrol_ManAut_2 : Int := 0;   // Bity przełączenia trybu pracy napędów / Bity przełączenia trybu pracy napędów Z5, Z6, Z7, Z8, Z9, Z10, Z11, Z12
         instLevelTank1 : Int := 0;   // Poziom zbiornik
         instLevelTank2 : Int := 0;   // Poziom zbiornik
         instLevelTank3 : Int := 0;   // Poziom zbiornik
         instLevelTank4 : Int := 0;   // Poziom zbiornik
         instPosition_Z10 : Real := 0.0;   // rezerwa / Zadawanie położenia Z10
         instClearFault1 : Int := 0;   // Bity kasowania alarmów napędów M1-M4, Z1 - Z12
         instSygSter_1 : Int := 2;   // rezerwa / Sygnały sterowania strategią pompownia - 0= wyłaczone, 1=dosilanie, 2=przetłaczanie,3=automat, 4=ręczne
         instSygSter_2 : Int := 1;   // Sygnały sterowania cyklem zbiorniki 0-wyłączone, 1=dobowy, 2=tygodniowy, 3=ręczne
         instCurrent_Inverter : Int := 0;   // Aktualny prądu falownika
         instHz_Inverter : Int := 0;   // Aktualne Hz na falowniku
      END_STRUCT;
      Pomiary : Struct
         instLevelSetFilling : Real := 550.0;   // Zadany poziom napełniania
         instLevelSetEmptying : Real := 10.0;   // Zadany poziom opróżniania
         instSetbarDN225_B6 : Real := 6.6;   // Zadany ciśnienie tłóczenia kierunek miasto, Modbus 40035
         instSetbarDN500_B5 : Real := 7.0;   // Zadana ciśnienie dosilania kierunek dosilanie "0" Modbus 40037
         instSetBarMinB9 : Real := 6.5;   // Zadawana dolna granica ciśnienia studnia "Granica" Modbus 40039
         instB5bar_act : Real;   // Aktualne ciśnienie zasilania z sieci
         instB6bar_act : Real;   // Aktualne ciśnienie DN225 tłoczny
         instB7bar_act : Real;   // Aktualne ciśnienie DN225 pompy
         instB8bar_act : Real;   // Aktualne ciśnienie ssoncy pomp (zab. Suchobieg)
         instPozitionZ10_act : Real;   // Aktualna pozycja zasuwy Z10
         instFlowDN225_act : Real;   // Przepływ DN225 aktualny MIASTO
         instFlowDN225_sum : Real;   // SUMA przepływu Dolna DN225
         instFlowDN500_act : Real;   // Przepływ DN500 (l/s) aktualny, zasilanie zbiorników, DOSILANIE, Modbus 40055
         instFlowDN500_sum : Real;   // SUMA przepływu Dolna DN500 Modbus 40057
      END_STRUCT;
      Godziny : Struct
         instHourStart_Filling : Int := 0;   // Godzina start napełniania
         instMinutStart_Filling : Int := 5;   // Minuta start napełniania
         instHourStop_Filling : Int := 17;   // Godzina stop napełniania
         instMinutStopt_Filling : Int := 0;   // Minuta stop napełniania
         instHourStart_City : Int := 18;   // Godzina start przetłaczanie miasto DN225
         instMinutStart_City : Int := 0;   // Minuty start przetłaczanie miasto DN225
         instHourStop_City : Int := 23;   // Godzina stop przetłaczanie miasto DN225
         instMinutStopt_City : Int := 59;   // Minuty stop przetłaczanie miasto DN225
         instHourStart_Replen : Int := 18;   // Godzina start przetłaczanie magistrala DN500
         instMinutStart_Replen : Int := 0;   // Minuty start przetłaczanie magistrala DN500
         instHourStop_Replen : Int := 23;   // Godzina stop przetłaczanie magistrala DN500
         instMinutStopt_Replen : Int := 59;   // Minuty stop przetłaczanie magistrala DN500
      END_STRUCT;
   END_VAR
BEGIN
END_DATA_BLOCK

DATA_BLOCK "dbHold_RRG"   // DB57
TITLE = Instancja danych serwera TCP
{ S7_Optimized_Access := 'FALSE' }
AUTHOR : rtecmer
VERSION : 0.1
// Instancja dla serwera Modbus TCP. Dane udostępniane i wpisywanedla PLC Zasuwy
// stored: AutoNumber true, DBAccessibleFromOPCUA true, IsOnlyStoredInLoadMemory false, IsWriteProtectedInAS false
   VAR
      actB5_bar_magistrala : Real;   // 4001-4002 Pomiar ciśnienia magistrala - dosilanie
      act_poziom_ZB1 : Real;   // 4003-4004 Pomiar poziom w zbiorniku
      act_poziom_ZB2 : Real;   // 4005-4006 Pomiar poziom w zbiorniku
      act_poziom_ZB3 : Real;   // 4007-4008 Pomiar poziom w zbiorniku
      act_poziom_ZB4 : Real;   // 4009-4010 Pomiar poziom w zbiorniku
      act_przepływ_VF_Q2 : Real;   // 4011-4012 Aktualny przepływ VF
      "act_przepływ-VR_Q2" : Real;   // 4013-4014 Aktualny przepływ VR wsteczny
      sum_przepływ_Q2 : Real;   // 4015-4016
      status_Z1 : Word;   // 4017
      status_Z2 : Word;   // 4018
      status_Z3 : Word;   // 4019
      status_Z4 : Word;   // 4020
      status_Z5 : Word;   // 4021
      status_Z6 : Word;   // 4022
      status_Z7 : Word;   // 4023
      status_Z8 : Word;   // 4024
      status_Z9 : Word;   // 4025
      status_Z10 : Word;   // 4026
      status_przepływomierz_Q2 : Word;   // 4027 status przepływomierza DN500
      act_położenie_Z10 : Word;   // 4028 Położenie zasuwy Z10 [%]
      komunikacja_PLC : Word;   // 4029 Kontrola komunikacji PLC1 - PLC2 wartość 0 wysyłane do PLC1
      set_poziom_napełniania : Real;   // 4030 - 4031 wartość zadana poziomu napełniania
      set_poziom_opróżniania : Real := 30.0;   // 4032 - 4033 wartość zadana poziomu opróżniania
      set_res_bity_sterowania_napęami_1 : Word;   // 4034 bity sterowania napędami
      set_res_bity_sterowania_napęami_2 : Word;   // 4035 bity sterowania napędami
      set_res_bity_tryb_napędów_1 : Word;   // 4036 bity sterowania przełączaniem trybów pracy
      set_res_bity_tryb_napędów_2 : Word;   // 4037 bity sterowania przełączaniem trybów pracy
      reset_alarm_napędów : Word;   // 4038 bity kasowania alarmów napędów
      set_strategia_sterowania : Word;   // 4039 (Bit 53.0 - Wyłączony), (Bit 53.1 - Dosilanie), (Bit 53.2 - Przetłączanie), (Bit 53.3 - Automat), (Bit 53.4 - Ręczne )
      set_sterowanie_cyklem : Word;   // 4040 (Bit 55.0 - Cykl wyłączony (Bit 55.1 - Cykl dobowy), (Bit 55.2 - Cykl tygodniowy), (Bit 55.3 - Cykl ręczny)
      set_położenie_Z10 : Word;   // 4041Położenie zasuwy Z10 [%]
      komunikacjaPLC : Word;   // 4042 kontrola komunikacji wysyłanie -> 0
      start_napełnianie : DTL := DTL#1970-01-01-23:55:00;   // 4043
      Stop_napełnianie : DTL := DTL#1970-01-01-16:00:00;
      Start_przetłaczanie_1 : DTL := DTL#1970-01-01-18:00:00;
      Stop_przetłaczanie_1 : DTL := DTL#1970-01-01-23:40:00;
      Start_dosilanie_1 : DTL := DTL#1970-01-01-18:00:00;
      Stop_dosilanie_1 : DTL := DTL#1970-01-01-23:40:00;
      Sending : Struct
         act_położenie_Z10 : Word := 40;   // Położenie zasuwy Z11 [%]
         set_poziom_napełniania : Real := 550.0;   // wartość zadana poziomu napełniania
         set_poziom_opróżniania : Real := 30.0;   // wartość zadana poziomu opróżniania
         set_res_bity_sterowania_napęami_1 : Word;   // bity sterowania napędami
         set_res_bity_sterowania_napęami_2 : Word;   // bity sterowania napędami
         set_res_bity_tryb_napędów_1 : Word;   // bity sterowania przełączaniem trybów pracy
         set_res_bity_tryb_napędów_2 : Word;   // bity sterowania przełączaniem trybów pracy
         rez_alarm_napędów : Word;   // bity kasowania alarmów napędów
         set_strategia_sterowania : Word;   // (Bit 53.0 - Wyłączony), (Bit 53.1 - Dosilanie), (Bit 53.2 - Przetłączanie), (Bit 53.3 - Automat), (Bit 53.4 - Ręczne )
         set_sterowanie_cyklem : Word;   // (Bit 55.0 - Cykl wyłączony (Bit 55.1 - Cykl dobowy), (Bit 55.2 - Cykl tygodniowy), (Bit 55.3 - Cykl ręczny)
         set_położenie_Z10 : Word;   // zadane położenie procentowe Z10
         komunikacjaPLC : Word;   // kontrola komunikacji wysyłanie -> 0
         set_magistrala_alarm_min_bar : Real := 6.5;   // wartość alarmowa awaria zasilania na magistrali B5
      END_STRUCT;
      SendingTimes : Struct
         start_napełnianie : DTL := DTL#1970-01-01-23:55:00;
         Stop_napełnianie : DTL := DTL#1970-01-01-16:00:00;
         Start_przetłaczanie_1 : DTL := DTL#1970-01-01-18:00:00;
         Stop_przetłaczanie_1 : DTL := DTL#1970-01-01-23:40:00;
         Start_dosilanie_1 : DTL := DTL#1970-01-01-18:00:00;
         Stop_dosilanie_1 : DTL := DTL#1970-01-01-23:40:00;
      END_STRUCT;
   END_VAR
BEGIN
END_DATA_BLOCK

DATA_BLOCK "dbHold_Sending_TCP"   // DB114
{ S7_Optimized_Access := 'FALSE' }
VERSION : 0.1
// stored: AutoNumber true, DBAccessibleFromOPCUA true, IsOnlyStoredInLoadMemory false, IsWriteProtectedInAS false
   VAR
      Sending_Hold : Struct
         set_poziom_napełniania : Real;   // wartość zadana poziomu napełniania
         set_poziom_opróżniania : Real;   // wartość zadana poziomu opróżniania
         set_bity_sterowania_napęami_1 : Word;   // bity sterowania napędami
         set_bity_sterowania_napęami_2 : Word;   // bity sterowania napędami
         set_bity_tryb_napędów_1 : Word;   // bity sterowania przełączaniem trybów pracy
         set_bity_tryb_napędów_2 : Word;   // bity sterowania przełączaniem trybów pracy
         rez_alarm_napędów : Word;   // bity kasowania alarmów napędów
         set_strategia_sterowania : Word;   // (Bit 53.0 - Wyłączony), (Bit 53.1 - Dosilanie), (Bit 53.2 - Przetłączanie), (Bit 53.3 - Automat), (Bit 53.4 - Ręczne )
         set_sterowanie_cyklem : Word;   // (Bit 55.0 - Cykl wyłączony (Bit 55.1 - Cykl dobowy), (Bit 55.2 - Cykl tygodniowy), (Bit 55.3 - Cykl ręczny)
         set_położenie_Z10 : Word;   // zadane położenie procentowe Z10
         komunikacjaPLC : Word := 1;   // kontrola komunikacji wysyłanie -> 1
         instHourStart_Filling : Int := 0;   // Godzina start napełniania
         instMinutStart_Filling : Int := 5;   // Minuta start napełniania
         instHourStop_Filling : Int := 17;   // Godzina stop napełniania
         instMinutStopt_Filling : Int := 0;   // Minuta stop napełniania
         instHourStart_City : Int := 18;   // Godzina start przetłaczanie miasto DN225
         instMinutStart_City : Int := 0;   // Minuty start przetłaczanie miasto DN225
         instHourStop_City : Int := 23;   // Godzina stop przetłaczanie miasto DN225
         instMinutStopt_City : Int := 59;   // Minuty stop przetłaczanie miasto DN225
         instHourStart_Replen : Int := 18;   // Godzina start przetłaczanie magistrala DN500
         instMinutStart_Replen : Int := 0;   // Minuty start przetłaczanie magistrala DN500
         instHourStop_Replen : Int := 23;   // Godzina stop przetłaczanie magistrala DN500
         instMinutStopt_Replen : Int := 59;   // Minuty stop przetłaczanie magistrala DN500
      END_STRUCT;
   END_VAR
BEGIN
END_DATA_BLOCK

DATA_BLOCK "ERR_Enum"   // DB105
{ S7_Optimized_Access := 'TRUE' }
VERSION : 0.1
// stored: AutoNumber false, DBAccessibleFromOPCUA true, IsOnlyStoredInLoadMemory false, IsRetainMemResEnabled false, IsWriteProtectedInAS false, MemoryReserve 0
   VAR
      GetErrorID : Array[0..27] of Word;
      SoftwareError { S7_SetPoint := 'True'} : "stt_ERR_Enum_SoftwareError";
      OB80 : Array[0..5] of Byte;
   END_VAR
BEGIN
   GetErrorID[0] := 16#2503;
   GetErrorID[1] := 16#2520;
   GetErrorID[2] := 16#2522;
   GetErrorID[3] := 16#2523;
   GetErrorID[4] := 16#2524;
   GetErrorID[5] := 16#2525;
   GetErrorID[6] := 16#2528;
   GetErrorID[7] := 16#2529;
   GetErrorID[8] := 16#252C;
   GetErrorID[9] := 16#2530;
   GetErrorID[10] := 16#2533;
   GetErrorID[11] := 16#2538;
   GetErrorID[12] := 16#2539;
   GetErrorID[13] := 16#253A;
   GetErrorID[14] := 16#253C;
   GetErrorID[15] := 16#253D;
   GetErrorID[16] := 16#253E;
   GetErrorID[17] := 16#253F;
   GetErrorID[18] := 16#2550;
   GetErrorID[19] := 16#2551;
   GetErrorID[20] := 16#2575;
   GetErrorID[21] := 16#2576;
   GetErrorID[22] := 16#2577;
   GetErrorID[23] := 16#25A0;
   GetErrorID[24] := 16#25A1;
   GetErrorID[25] := 16#25A2;
   GetErrorID[26] := 16#2942;
   GetErrorID[27] := 16#2943;
END_DATA_BLOCK

DATA_BLOCK "ERR_ErrorBufferFull"   // DB106
{ S7_Optimized_Access := 'TRUE' }
VERSION : 0.1
// stored: AutoNumber false, DBAccessibleFromOPCUA true, IsOnlyStoredInLoadMemory false, IsRetainMemResEnabled false, IsWriteProtectedInAS false, MemoryReserve 0
   VAR
      Error { S7_SetPoint := 'True'} : ErrorStruct;
   END_VAR
   VAR RETAIN
      SoftwareError { S7_SetPoint := 'True'} : Array[0..4] of "stt_ERR_SoftwareError";
      GetError { S7_SetPoint := 'True'} : Array[0..27] of "stt_ERR_GetError";
      CounterDiagStatusUpdate : UInt;
   END_VAR
BEGIN
END_DATA_BLOCK

DATA_BLOCK "ERR_ErrorOB"   // DB107
{ S7_Optimized_Access := 'TRUE' }
VERSION : 0.1
// stored: AutoNumber false, DBAccessibleFromOPCUA true, IsOnlyStoredInLoadMemory false, IsRetainMemResEnabled false, IsWriteProtectedInAS false, MemoryReserve 0
   VAR RETAIN
      OB80 { S7_SetPoint := 'True'} : Array[0..5] of "stt_ERR_OB80";
   END_VAR
BEGIN
END_DATA_BLOCK

DATA_BLOCK "V_ErrorOB"   // DB108
{ S7_Optimized_Access := 'TRUE' }
VERSION : 0.1
// stored: AutoNumber false, DBAccessibleFromOPCUA true, IsOnlyStoredInLoadMemory false, IsRetainMemResEnabled false, IsWriteProtectedInAS false, MemoryReserve 0
   VAR
      StartUp { S7_SetPoint := 'True'} : "stt_ERR_StartUpOB";   // //Error read in OB100
      OB80 : Bool;   // //Executed OB80 Time error interrupt
      ResetErrorOB : Bool;   // //Variable connected with button in web site
   END_VAR
BEGIN
END_DATA_BLOCK

DATA_BLOCK "V_SoftwareError"   // DB109
{ S7_Optimized_Access := 'TRUE' }
VERSION : 0.1
// stored: AutoNumber false, DBAccessibleFromOPCUA true, IsOnlyStoredInLoadMemory false, IsRetainMemResEnabled false, IsWriteProtectedInAS false, MemoryReserve 0
   VAR
      SoftwareFunctions : Bool;   // //Error is appear in called function
      GetErrorFunction : Bool;   // //Function GET_ERROR() return error
      DiagnosticBuffer : Bool;   // //Error is appear in diagnostic buffer
      ResetErrorSoftware : Bool;   // //Variable connected with button in web site
   END_VAR
BEGIN
END_DATA_BLOCK

DATA_BLOCK "V_LED"   // DB110
{ S7_Optimized_Access := 'TRUE' }
VERSION : 0.1
// stored: AutoNumber false, DBAccessibleFromOPCUA true, IsOnlyStoredInLoadMemory false, IsRetainMemResEnabled false, IsWriteProtectedInAS false, MemoryReserve 0
   VAR
      LED : Array[1..6] of Int;   // //Status for each module LED
   END_VAR
BEGIN
END_DATA_BLOCK

ORGANIZATION_BLOCK "OB1"   // OB1, LAD, ProgramCycle
TITLE = Głowny blok
{ S7_Optimized_Access := 'TRUE' }
AUTHOR : RTecmer
VERSION : 0.1
// stored: AutoNumber true, IsIECCheckEnabled false, SetENOAutomatically false
   VAR_INPUT
      Initial_Call : Bool;   // Initial call of this OB
      Remanence : Bool;   // =True, if remanent data are available
   END_VAR
   VAR_TEMP
      tempWatchDog_HMI : Int;
   END_VAR
   VAR_TEMP   // added for the SCL form of the ladder/FBD networks
      _w1 : Bool;
      _w2 : Bool;
   END_VAR
BEGIN

REGION Network 2: Zegart RTC
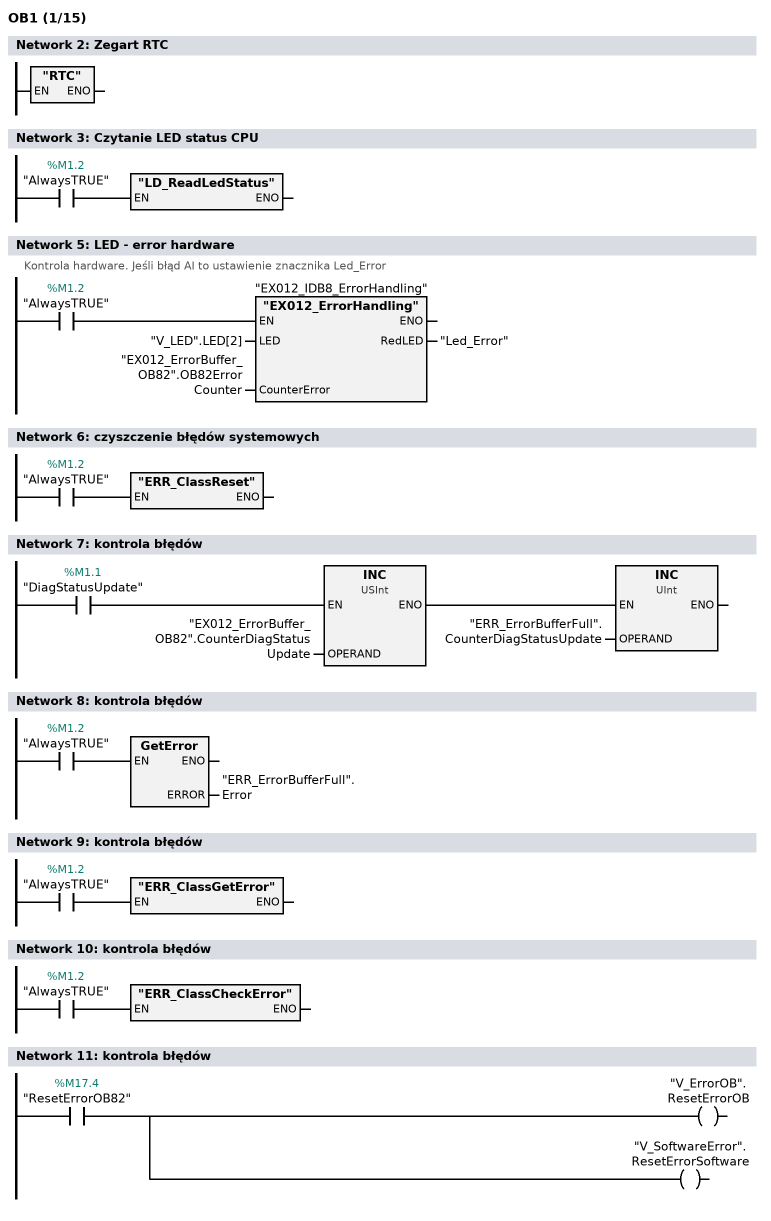
   RUNG wire#powerrail
      "RTC"()
   END_RUNG
   // the same network as SCL:
   "RTC"();
END_REGION

REGION Network 3: Czytanie LED status CPU
   RUNG wire#powerrail
      Contact( "AlwaysTRUE" )
      "LD_ReadLedStatus"()
   END_RUNG
   // the same network as SCL:
   IF "AlwaysTRUE" THEN "LD_ReadLedStatus"(); END_IF;
END_REGION

REGION Network 4 (SCL): LED kontrola RUN
   // Przekazanie  stanu LED 1 CPU
   "DB31_HMI_AreaPointer".getPLCMode := "V_LED".LED[1];
END_REGION

REGION Network 5: LED - error hardware
   // Kontrola hardware. Jeśli błąd AI to ustawienie znacznika Led_Error
   RUNG wire#powerrail
      Contact( "AlwaysTRUE" )
      "EX012_IDB8_ErrorHandling"(LED := "V_LED".LED[2], CounterError := "EX012_ErrorBuffer_OB82".OB82ErrorCounter, RedLED => "Led_Error")
   END_RUNG
   // the same network as SCL:
   IF "AlwaysTRUE" THEN
       "EX012_IDB8_ErrorHandling"(LED := "V_LED".LED[2],   // "EX012_ErrorHandling"
                               CounterError := "EX012_ErrorBuffer_OB82".OB82ErrorCounter,
                               RedLED => "Led_Error");
   END_IF;
END_REGION

REGION Network 6: czyszczenie błędów systemowych
   RUNG wire#powerrail
      Contact( "AlwaysTRUE" )
      "ERR_ClassReset"()
   END_RUNG
   // the same network as SCL:
   IF "AlwaysTRUE" THEN "ERR_ClassReset"(); END_IF;
END_REGION

REGION Network 7: kontrola błędów
   RUNG wire#powerrail
      Contact( "DiagStatusUpdate" )
      { S7_Templates := "DestType := USInt" } Inc( "EX012_ErrorBuffer_OB82".CounterDiagStatusUpdate )
      { S7_Templates := "DestType := UInt" } Inc( "ERR_ErrorBufferFull".CounterDiagStatusUpdate )
   END_RUNG
   // the same network as SCL:
   IF "DiagStatusUpdate" THEN
       "EX012_ErrorBuffer_OB82".CounterDiagStatusUpdate := "EX012_ErrorBuffer_OB82".CounterDiagStatusUpdate + 1;
       "ERR_ErrorBufferFull".CounterDiagStatusUpdate := "ERR_ErrorBufferFull".CounterDiagStatusUpdate + 1;
   END_IF;
END_REGION

REGION Network 8: kontrola błędów
   // no SCL statement known for GetError: written as a call
   IF "AlwaysTRUE" THEN GetError(error => "ERR_ErrorBufferFull".Error); END_IF;
END_REGION

REGION Network 9: kontrola błędów
   RUNG wire#powerrail
      Contact( "AlwaysTRUE" )
      "ERR_ClassGetError"()
   END_RUNG
   // the same network as SCL:
   IF "AlwaysTRUE" THEN "ERR_ClassGetError"(); END_IF;
END_REGION

REGION Network 10: kontrola błędów
   RUNG wire#powerrail
      Contact( "AlwaysTRUE" )
      "ERR_ClassCheckError"()
   END_RUNG
   // the same network as SCL:
   IF "AlwaysTRUE" THEN "ERR_ClassCheckError"(); END_IF;
END_REGION

REGION Network 11: kontrola błędów
   RUNG wire#powerrail
      Contact( "ResetErrorOB82" )
      wire#w1
      Coil( "V_ErrorOB".ResetErrorOB )
   END_RUNG
   RUNG wire#w1
      Coil( "V_SoftwareError".ResetErrorSoftware )
   END_RUNG
   // the same network as SCL:
   "V_ErrorOB".ResetErrorOB := "ResetErrorOB82";
   "V_SoftwareError".ResetErrorSoftware := "ResetErrorOB82";
END_REGION

REGION Network 12: Kasowanie alarmów napędów z poziomu SCADA
   // Komunikacja Modbus RTU - MT101
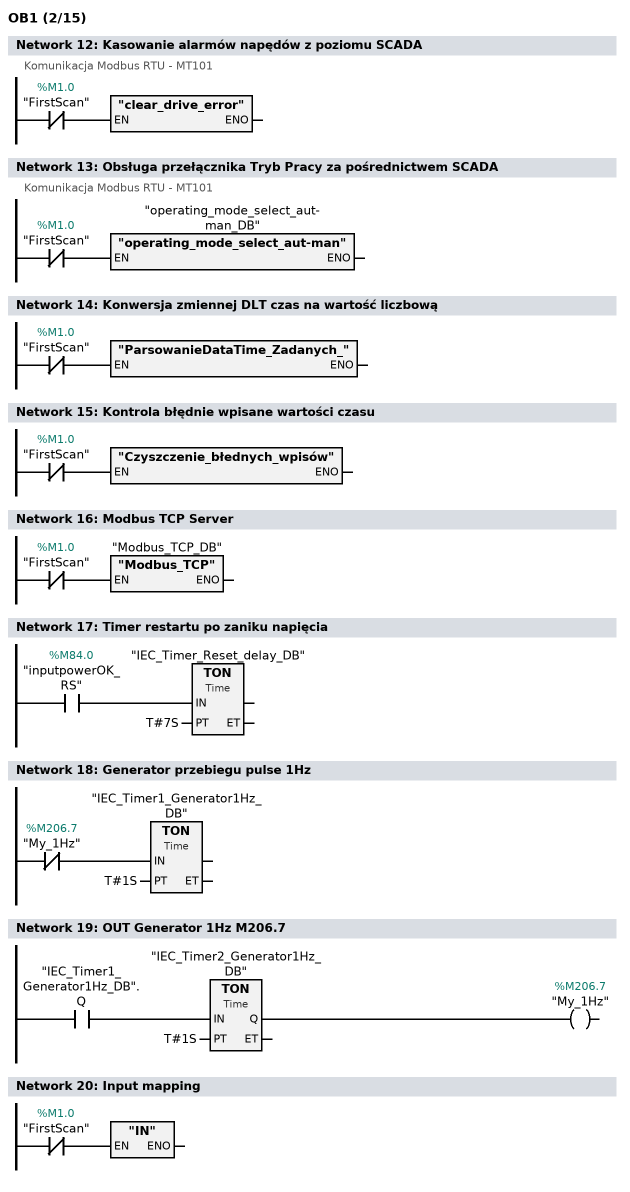
   RUNG wire#powerrail
      I_Contact( "FirstScan" )
      "clear_drive_error"()
   END_RUNG
   // the same network as SCL:
   IF NOT "FirstScan" THEN "clear_drive_error"(); END_IF;
END_REGION

REGION Network 13: Obsługa przełącznika Tryb Pracy za pośrednictwem SCADA
   // Komunikacja Modbus RTU - MT101
   RUNG wire#powerrail
      I_Contact( "FirstScan" )
      "operating_mode_select_aut-man_DB"()
   END_RUNG
   // the same network as SCL:
   IF NOT "FirstScan" THEN
       "operating_mode_select_aut-man_DB"();   // "operating_mode_select_aut-man"
   END_IF;
END_REGION

REGION Network 14: Konwersja zmiennej DLT czas na wartość liczbową
   RUNG wire#powerrail
      I_Contact( "FirstScan" )
      "ParsowanieDataTime_Zadanych_"()
   END_RUNG
   // the same network as SCL:
   IF NOT "FirstScan" THEN "ParsowanieDataTime_Zadanych_"(); END_IF;
END_REGION

REGION Network 15: Kontrola błędnie wpisane wartości czasu
   RUNG wire#powerrail
      I_Contact( "FirstScan" )
      "Czyszczenie_błednych_wpisów"()
   END_RUNG
   // the same network as SCL:
   IF NOT "FirstScan" THEN "Czyszczenie_błednych_wpisów"(); END_IF;
END_REGION

REGION Network 16: Modbus TCP Server
   RUNG wire#powerrail
      I_Contact( "FirstScan" )
      "Modbus_TCP_DB"()
   END_RUNG
   // the same network as SCL:
   IF NOT "FirstScan" THEN
       "Modbus_TCP_DB"();   // "Modbus_TCP"
   END_IF;
END_REGION

REGION Network 17: Timer restartu po zaniku napięcia
   RUNG wire#powerrail
      Contact( "inputpowerOK_RS" )
      { S7_Templates := "time_type := Time" } "IEC_Timer_Reset_delay_DB".TON(pt := T#7S, et =>)
   END_RUNG
   // the same network as SCL:
   "IEC_Timer_Reset_delay_DB".TON(IN := "inputpowerOK_RS", PT := T#7S);
END_REGION

REGION Network 18: Generator przebiegu pulse 1Hz
   RUNG wire#powerrail
      I_Contact( "My_1Hz" )
      { S7_Templates := "time_type := Time" } "IEC_Timer1_Generator1Hz_DB".TON(pt := T#1S, et =>)
   END_RUNG
   // the same network as SCL:
   "IEC_Timer1_Generator1Hz_DB".TON(IN := NOT "My_1Hz", PT := T#1S);
END_REGION

REGION Network 19: OUT Generator 1Hz M206.7
   RUNG wire#powerrail
      Contact( "IEC_Timer1_Generator1Hz_DB".Q )
      { S7_Templates := "time_type := Time" } "IEC_Timer2_Generator1Hz_DB".TON(pt := T#1S, et =>)
      Coil( "My_1Hz" )
   END_RUNG
   // the same network as SCL:
   "IEC_Timer2_Generator1Hz_DB".TON(IN := "IEC_Timer1_Generator1Hz_DB".Q, PT := T#1S);
   "My_1Hz" := "IEC_Timer2_Generator1Hz_DB".Q;
END_REGION

REGION Network 20: Input mapping
   RUNG wire#powerrail
      I_Contact( "FirstScan" )
      "IN"()
   END_RUNG
   // the same network as SCL:
   IF NOT "FirstScan" THEN "IN"(); END_IF;
END_REGION

REGION Network 21: filtr kolmana - analogi
   // eliminacja szybkozmiennych zakłóceń
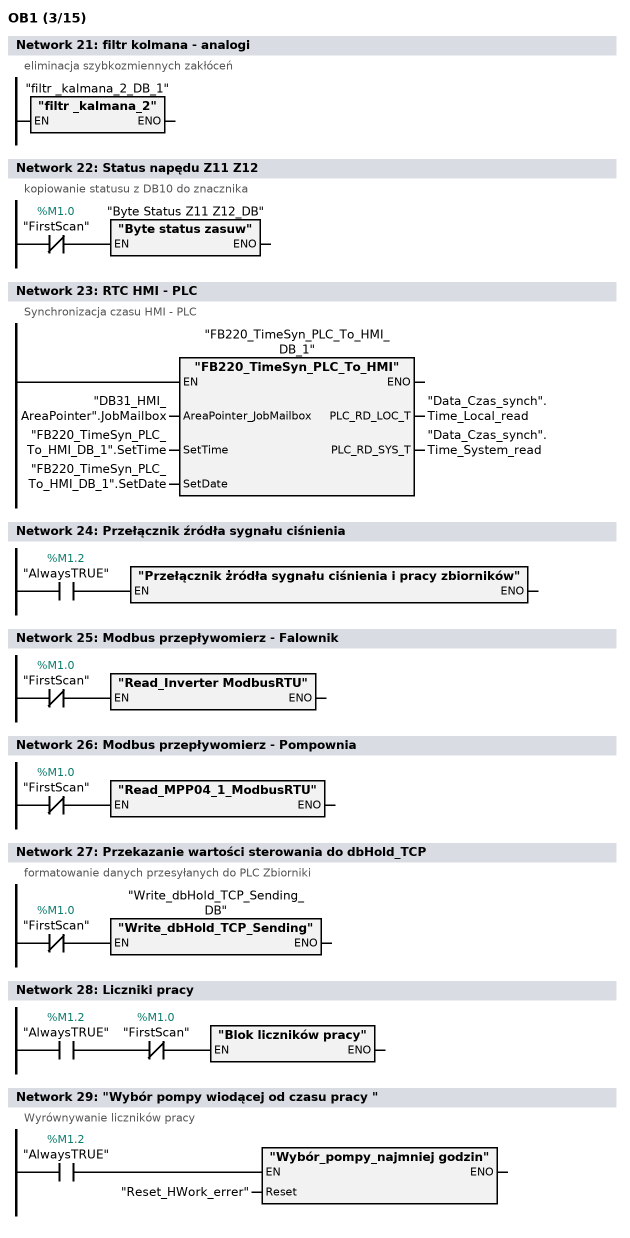
   RUNG wire#powerrail
      "filtr _kalmana_2_DB_1"()
   END_RUNG
   // the same network as SCL:
   "filtr _kalmana_2_DB_1"();   // "filtr _kalmana_2"
END_REGION

REGION Network 22: Status napędu Z11 Z12
   // kopiowanie statusu z DB10 do znacznika
   RUNG wire#powerrail
      I_Contact( "FirstScan" )
      "Byte Status Z11 Z12_DB"()
   END_RUNG
   // the same network as SCL:
   IF NOT "FirstScan" THEN
       "Byte Status Z11 Z12_DB"();   // "Byte status zasuw"
   END_IF;
END_REGION

REGION Network 23: RTC HMI - PLC
   // Synchronizacja czasu HMI - PLC
   RUNG wire#powerrail
      "FB220_TimeSyn_PLC_To_HMI_DB_1"(AreaPointer_JobMailbox := "DB31_HMI_AreaPointer".JobMailbox, SetTime := "FB220_TimeSyn_PLC_To_HMI_DB_1".SetTime, SetDate := "FB220_TimeSyn_PLC_To_HMI_DB_1".SetDate, PLC_RD_LOC_T => "Data_Czas_synch".Time_Local_read, PLC_RD_SYS_T => "Data_Czas_synch".Time_System_read)
   END_RUNG
   // the same network as SCL:
   "FB220_TimeSyn_PLC_To_HMI_DB_1"(AreaPointer_JobMailbox := "DB31_HMI_AreaPointer".JobMailbox,   // "FB220_TimeSyn_PLC_To_HMI"
                           SetTime := "FB220_TimeSyn_PLC_To_HMI_DB_1".SetTime,
                           SetDate := "FB220_TimeSyn_PLC_To_HMI_DB_1".SetDate,
                           PLC_RD_LOC_T => "Data_Czas_synch".Time_Local_read,
                           PLC_RD_SYS_T => "Data_Czas_synch".Time_System_read);
END_REGION

REGION Network 24: Przełącznik źródła sygnału ciśnienia
   RUNG wire#powerrail
      Contact( "AlwaysTRUE" )
      "Przełącznik żródła sygnału ciśnienia i pracy zbiorników"()
   END_RUNG
   // the same network as SCL:
   IF "AlwaysTRUE" THEN "Przełącznik żródła sygnału ciśnienia i pracy zbiorników"(); END_IF;
END_REGION

REGION Network 25: Modbus przepływomierz - Falownik
   RUNG wire#powerrail
      I_Contact( "FirstScan" )
      "Read_Inverter ModbusRTU"()
   END_RUNG
   // the same network as SCL:
   IF NOT "FirstScan" THEN "Read_Inverter ModbusRTU"(); END_IF;
END_REGION

REGION Network 26: Modbus przepływomierz - Pompownia
   RUNG wire#powerrail
      I_Contact( "FirstScan" )
      "Read_MPP04_1_ModbusRTU"()
   END_RUNG
   // the same network as SCL:
   IF NOT "FirstScan" THEN "Read_MPP04_1_ModbusRTU"(); END_IF;
END_REGION

REGION Network 27: Przekazanie wartości sterowania do dbHold_TCP
   // formatowanie danych przesyłanych do PLC Zbiorniki
   RUNG wire#powerrail
      I_Contact( "FirstScan" )
      "Write_dbHold_TCP_Sending_DB"()
   END_RUNG
   // the same network as SCL:
   IF NOT "FirstScan" THEN
       "Write_dbHold_TCP_Sending_DB"();   // "Write_dbHold_TCP_Sending"
   END_IF;
END_REGION

REGION Network 28: Liczniki pracy
   RUNG wire#powerrail
      Contact( "AlwaysTRUE" )
      I_Contact( "FirstScan" )
      "Blok liczników pracy"()
   END_RUNG
   // the same network as SCL:
   IF "AlwaysTRUE" AND NOT "FirstScan" THEN "Blok liczników pracy"(); END_IF;
END_REGION

REGION Network 29: "Wybór pompy wiodącej od czasu pracy "
   // Wyrównywanie liczników pracy
   RUNG wire#powerrail
      Contact( "AlwaysTRUE" )
      "Wybór_pompy_najmniej godzin"(Reset := "Reset_HWork_errer")
   END_RUNG
   // the same network as SCL:
   IF "AlwaysTRUE" THEN "Wybór_pompy_najmniej godzin"(Reset := "Reset_HWork_errer"); END_IF;
END_REGION

REGION Network 30: Obsługa błędów Modbus RTU
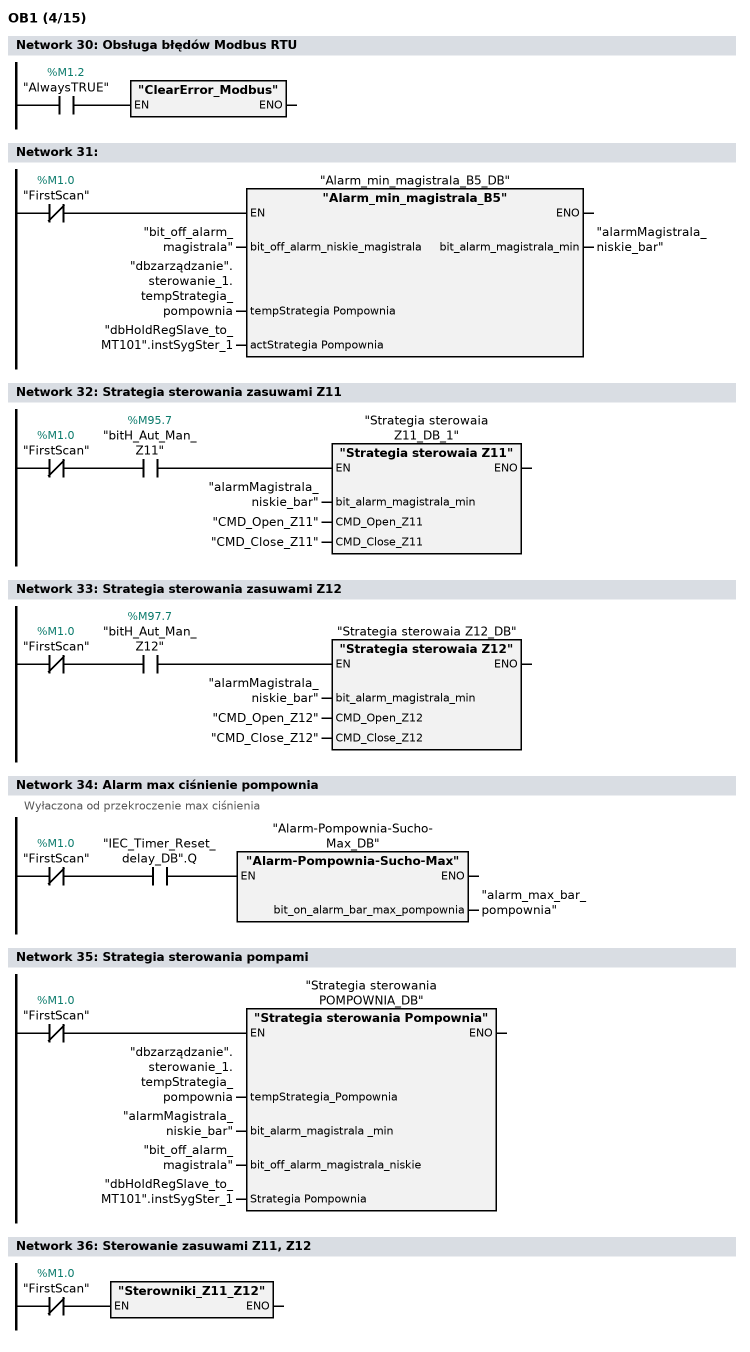
   RUNG wire#powerrail
      Contact( "AlwaysTRUE" )
      "ClearError_Modbus"()
   END_RUNG
   // the same network as SCL:
   IF "AlwaysTRUE" THEN "ClearError_Modbus"(); END_IF;
END_REGION

REGION Network 31
   RUNG wire#powerrail
      I_Contact( "FirstScan" )
      "Alarm_min_magistrala_B5_DB"(bit_off_alarm_niskie_magistrala := "bit_off_alarm_magistrala", "tempStrategia Pompownia" := "dbzarządzanie".sterowanie_1.tempStrategia_pompownia, "actStrategia Pompownia" := "dbHoldRegSlave_to_MT101".instSygSter_1, bit_alarm_magistrala_min => "alarmMagistrala_niskie_bar")
   END_RUNG
   // the same network as SCL:
   IF NOT "FirstScan" THEN
       "Alarm_min_magistrala_B5_DB"(bit_off_alarm_niskie_magistrala := "bit_off_alarm_magistrala",   // "Alarm_min_magistrala_B5"
                               "tempStrategia Pompownia" := "dbzarządzanie".sterowanie_1.tempStrategia_pompownia,
                               "actStrategia Pompownia" := "dbHoldRegSlave_to_MT101".instSygSter_1,
                               bit_alarm_magistrala_min => "alarmMagistrala_niskie_bar");
   END_IF;
END_REGION

REGION Network 32: Strategia sterowania zasuwami Z11
   RUNG wire#powerrail
      I_Contact( "FirstScan" )
      Contact( "bitH_Aut_Man_Z11" )
      "Strategia sterowaia Z11_DB_1"(bit_alarm_magistrala_min := "alarmMagistrala_niskie_bar", CMD_Open_Z11 := "CMD_Open_Z11", CMD_Close_Z11 := "CMD_Close_Z11")
   END_RUNG
   // the same network as SCL:
   IF NOT "FirstScan" AND "bitH_Aut_Man_Z11" THEN
       "Strategia sterowaia Z11_DB_1"(bit_alarm_magistrala_min := "alarmMagistrala_niskie_bar",   // "Strategia sterowaia Z11"
                               CMD_Open_Z11 := "CMD_Open_Z11",
                               CMD_Close_Z11 := "CMD_Close_Z11");
   END_IF;
END_REGION

REGION Network 33: Strategia sterowania zasuwami Z12
   RUNG wire#powerrail
      I_Contact( "FirstScan" )
      Contact( "bitH_Aut_Man_Z12" )
      "Strategia sterowaia Z12_DB"(bit_alarm_magistrala_min := "alarmMagistrala_niskie_bar", CMD_Open_Z12 := "CMD_Open_Z12", CMD_Close_Z12 := "CMD_Close_Z12")
   END_RUNG
   // the same network as SCL:
   IF NOT "FirstScan" AND "bitH_Aut_Man_Z12" THEN
       "Strategia sterowaia Z12_DB"(bit_alarm_magistrala_min := "alarmMagistrala_niskie_bar",   // "Strategia sterowaia Z12"
                               CMD_Open_Z12 := "CMD_Open_Z12",
                               CMD_Close_Z12 := "CMD_Close_Z12");
   END_IF;
END_REGION

REGION Network 34: Alarm max ciśnienie pompownia
   // Wyłaczona od przekroczenie max ciśnienia
   RUNG wire#powerrail
      I_Contact( "FirstScan" )
      Contact( "IEC_Timer_Reset_delay_DB".Q )
      "Alarm-Pompownia-Sucho-Max_DB"(bit_on_alarm_bar_max_pompownia => "alarm_max_bar_pompownia")
   END_RUNG
   // the same network as SCL:
   IF NOT "FirstScan" AND "IEC_Timer_Reset_delay_DB".Q THEN
       "Alarm-Pompownia-Sucho-Max_DB"(bit_on_alarm_bar_max_pompownia => "alarm_max_bar_pompownia");   // "Alarm-Pompownia-Sucho-Max"
   END_IF;
END_REGION

REGION Network 35: Strategia sterowania pompami
   RUNG wire#powerrail
      I_Contact( "FirstScan" )
      "Strategia sterowania POMPOWNIA_DB"(tempStrategia_Pompownia := "dbzarządzanie".sterowanie_1.tempStrategia_pompownia, "bit_alarm_magistrala _min" := "alarmMagistrala_niskie_bar", bit_off_alarm_magistrala_niskie := "bit_off_alarm_magistrala", "Strategia Pompownia" := "dbHoldRegSlave_to_MT101".instSygSter_1)
   END_RUNG
   // the same network as SCL:
   IF NOT "FirstScan" THEN
       "Strategia sterowania POMPOWNIA_DB"(tempStrategia_Pompownia := "dbzarządzanie".sterowanie_1.tempStrategia_pompownia,   // "Strategia sterowania Pompownia"
                               "bit_alarm_magistrala _min" := "alarmMagistrala_niskie_bar",
                               bit_off_alarm_magistrala_niskie := "bit_off_alarm_magistrala",
                               "Strategia Pompownia" := "dbHoldRegSlave_to_MT101".instSygSter_1);
   END_IF;
END_REGION

REGION Network 36: Sterowanie zasuwami Z11, Z12
   RUNG wire#powerrail
      I_Contact( "FirstScan" )
      "Sterowniki_Z11_Z12"()
   END_RUNG
   // the same network as SCL:
   IF NOT "FirstScan" THEN "Sterowniki_Z11_Z12"(); END_IF;
END_REGION

REGION Network 37: Konwerter parametrów z falownika
   // funkcja wylicza wartości pobrane z falownika protokołem Modbus RTU
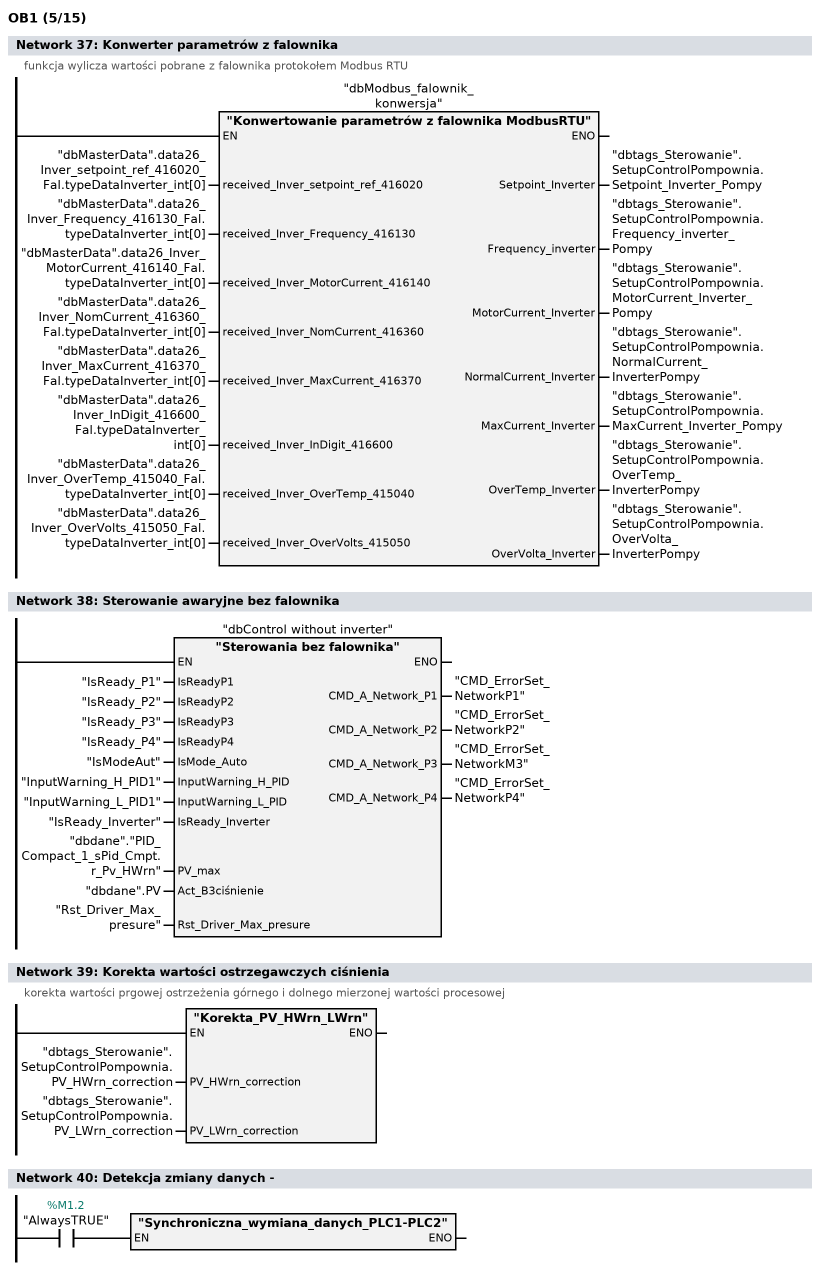
   RUNG wire#powerrail
      "dbModbus_falownik_konwersja"(received_Inver_setpoint_ref_416020 := "dbMasterData".data26_Inver_setpoint_ref_416020_Fal.typeDataInverter_int[0], received_Inver_Frequency_416130 := "dbMasterData".data26_Inver_Frequency_416130_Fal.typeDataInverter_int[0], received_Inver_MotorCurrent_416140 := "dbMasterData".data26_Inver_MotorCurrent_416140_Fal.typeDataInverter_int[0], received_Inver_NomCurrent_416360 := "dbMasterData".data26_Inver_NomCurrent_416360_Fal.typeDataInverter_int[0], received_Inver_MaxCurrent_416370 := "dbMasterData".data26_Inver_MaxCurrent_416370_Fal.typeDataInverter_int[0], received_Inver_InDigit_416600 := "dbMasterData".data26_Inver_InDigit_416600_Fal.typeDataInverter_int[0], received_Inver_OverTemp_415040 := "dbMasterData".data26_Inver_OverTemp_415040_Fal.typeDataInverter_int[0], received_Inver_OverVolts_415050 := "dbMasterData".data26_Inver_OverVolts_415050_Fal.typeDataInverter_int[0], Setpoint_Inverter => "dbtags_Sterowanie".SetupControlPompownia.Setpoint_Inverter_Pompy, Frequency_inverter => "dbtags_Sterowanie".SetupControlPompownia.Frequency_inverter_Pompy, MotorCurrent_Inverter => "dbtags_Sterowanie".SetupControlPompownia.MotorCurrent_Inverter_Pompy, NormalCurrent_Inverter => "dbtags_Sterowanie".SetupControlPompownia.NormalCurrent_InverterPompy, MaxCurrent_Inverter => "dbtags_Sterowanie".SetupControlPompownia.MaxCurrent_Inverter_Pompy, OverTemp_Inverter => "dbtags_Sterowanie".SetupControlPompownia.OverTemp_InverterPompy, OverVolta_Inverter => "dbtags_Sterowanie".SetupControlPompownia.OverVolta_InverterPompy)
   END_RUNG
   // the same network as SCL:
   "dbModbus_falownik_konwersja"(received_Inver_setpoint_ref_416020 := "dbMasterData".data26_Inver_setpoint_ref_416020_Fal.typeDataInverter_int[0],   // "Konwertowanie parametrów z falownika ModbusRTU"
                           received_Inver_Frequency_416130 := "dbMasterData".data26_Inver_Frequency_416130_Fal.typeDataInverter_int[0],
                           received_Inver_MotorCurrent_416140 := "dbMasterData".data26_Inver_MotorCurrent_416140_Fal.typeDataInverter_int[0],
                           received_Inver_NomCurrent_416360 := "dbMasterData".data26_Inver_NomCurrent_416360_Fal.typeDataInverter_int[0],
                           received_Inver_MaxCurrent_416370 := "dbMasterData".data26_Inver_MaxCurrent_416370_Fal.typeDataInverter_int[0],
                           received_Inver_InDigit_416600 := "dbMasterData".data26_Inver_InDigit_416600_Fal.typeDataInverter_int[0],
                           received_Inver_OverTemp_415040 := "dbMasterData".data26_Inver_OverTemp_415040_Fal.typeDataInverter_int[0],
                           received_Inver_OverVolts_415050 := "dbMasterData".data26_Inver_OverVolts_415050_Fal.typeDataInverter_int[0],
                           Setpoint_Inverter => "dbtags_Sterowanie".SetupControlPompownia.Setpoint_Inverter_Pompy,
                           Frequency_inverter => "dbtags_Sterowanie".SetupControlPompownia.Frequency_inverter_Pompy,
                           MotorCurrent_Inverter => "dbtags_Sterowanie".SetupControlPompownia.MotorCurrent_Inverter_Pompy,
                           NormalCurrent_Inverter => "dbtags_Sterowanie".SetupControlPompownia.NormalCurrent_InverterPompy,
                           MaxCurrent_Inverter => "dbtags_Sterowanie".SetupControlPompownia.MaxCurrent_Inverter_Pompy,
                           OverTemp_Inverter => "dbtags_Sterowanie".SetupControlPompownia.OverTemp_InverterPompy,
                           OverVolta_Inverter => "dbtags_Sterowanie".SetupControlPompownia.OverVolta_InverterPompy);
END_REGION

REGION Network 38: Sterowanie awaryjne bez falownika
   RUNG wire#powerrail
      "dbControl without inverter"(IsReadyP1 := "IsReady_P1", IsReadyP2 := "IsReady_P2", IsReadyP3 := "IsReady_P3", IsReadyP4 := "IsReady_P4", IsMode_Auto := "IsModeAut", InputWarning_H_PID := "InputWarning_H_PID1", InputWarning_L_PID := "InputWarning_L_PID1", IsReady_Inverter := "IsReady_Inverter", PV_max := "dbdane"."PID_Compact_1_sPid_Cmpt.r_Pv_HWrn", Act_B3ciśnienie := "dbdane".PV, Rst_Driver_Max_presure := "Rst_Driver_Max_presure", CMD_A_Network_P1 => "CMD_ErrorSet_NetworkP1", CMD_A_Network_P2 => "CMD_ErrorSet_NetworkP2", CMD_A_Network_P3 => "CMD_ErrorSet_NetworkM3", CMD_A_Network_P4 => "CMD_ErrorSet_NetworkP4")
   END_RUNG
   // the same network as SCL:
   "dbControl without inverter"(IsReadyP1 := "IsReady_P1",   // "Sterowania bez falownika"
                           IsReadyP2 := "IsReady_P2",
                           IsReadyP3 := "IsReady_P3",
                           IsReadyP4 := "IsReady_P4",
                           IsMode_Auto := "IsModeAut",
                           InputWarning_H_PID := "InputWarning_H_PID1",
                           InputWarning_L_PID := "InputWarning_L_PID1",
                           IsReady_Inverter := "IsReady_Inverter",
                           PV_max := "dbdane"."PID_Compact_1_sPid_Cmpt.r_Pv_HWrn",
                           Act_B3ciśnienie := "dbdane".PV,
                           Rst_Driver_Max_presure := "Rst_Driver_Max_presure",
                           CMD_A_Network_P1 => "CMD_ErrorSet_NetworkP1",
                           CMD_A_Network_P2 => "CMD_ErrorSet_NetworkP2",
                           CMD_A_Network_P3 => "CMD_ErrorSet_NetworkM3",
                           CMD_A_Network_P4 => "CMD_ErrorSet_NetworkP4");
END_REGION

REGION Network 39: Korekta wartości ostrzegawczych ciśnienia
   // korekta wartości prgowej ostrzeżenia górnego i dolnego mierzonej wartości procesowej
   RUNG wire#powerrail
      "Korekta_PV_HWrn_LWrn"(PV_HWrn_correction := "dbtags_Sterowanie".SetupControlPompownia.PV_HWrn_correction, PV_LWrn_correction := "dbtags_Sterowanie".SetupControlPompownia.PV_LWrn_correction)
   END_RUNG
   // the same network as SCL:
   "Korekta_PV_HWrn_LWrn"(PV_HWrn_correction := "dbtags_Sterowanie".SetupControlPompownia.PV_HWrn_correction,
                          PV_LWrn_correction := "dbtags_Sterowanie".SetupControlPompownia.PV_LWrn_correction);
END_REGION

REGION Network 40: Detekcja zmiany danych -
   RUNG wire#powerrail
      Contact( "AlwaysTRUE" )
      "Synchroniczna_wymiana_danych_PLC1-PLC2"()
   END_RUNG
   // the same network as SCL:
   IF "AlwaysTRUE" THEN "Synchroniczna_wymiana_danych_PLC1-PLC2"(); END_IF;
END_REGION

REGION Network 42: Sterowanie napędami pomp
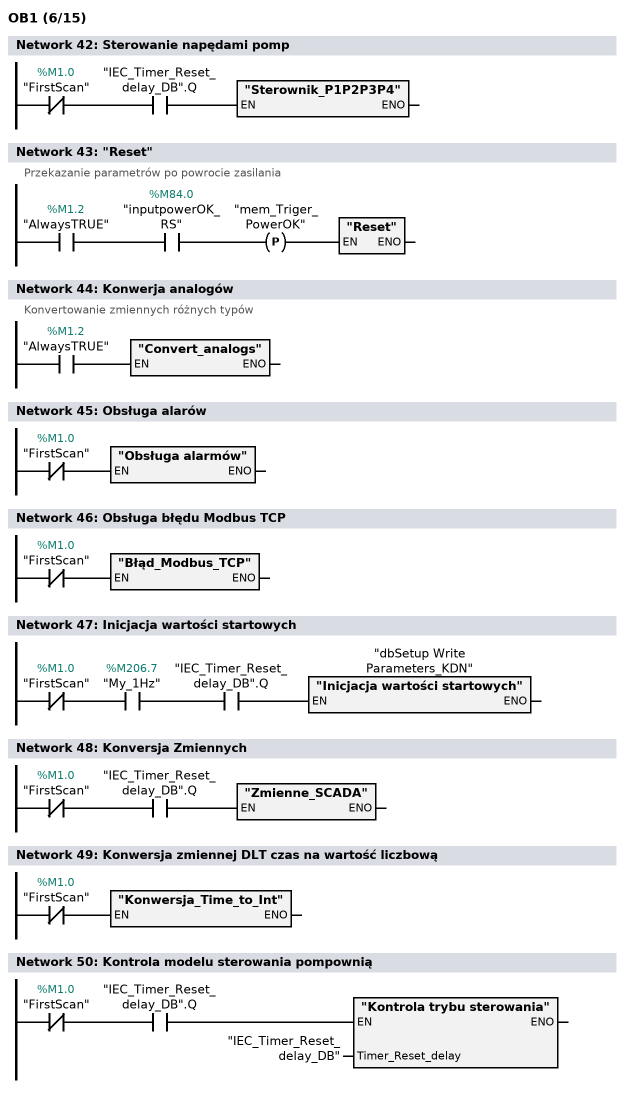
   RUNG wire#powerrail
      I_Contact( "FirstScan" )
      Contact( "IEC_Timer_Reset_delay_DB".Q )
      "Sterownik_P1P2P3P4"()
   END_RUNG
   // the same network as SCL:
   IF NOT "FirstScan" AND "IEC_Timer_Reset_delay_DB".Q THEN "Sterownik_P1P2P3P4"(); END_IF;
END_REGION

REGION Network 43: "Reset"
   // Przekazanie parametrów po powrocie zasilania
   RUNG wire#powerrail
      Contact( "AlwaysTRUE" )
      Contact( "inputpowerOK_RS" )
      P_Trig( "mem_Triger_PowerOK" )
      "Reset"()
   END_RUNG
   // the same network as SCL:
   #_w1 := "AlwaysTRUE" AND "inputpowerOK_RS";
   #_w2 := #_w1 AND NOT "mem_Triger_PowerOK";   // rising edge
   "mem_Triger_PowerOK" := #_w1;
   IF #_w2 THEN "Reset"(); END_IF;
END_REGION

REGION Network 44: Konwerja analogów
   // Konvertowanie zmiennych różnych typów
   RUNG wire#powerrail
      Contact( "AlwaysTRUE" )
      "Convert_analogs"()
   END_RUNG
   // the same network as SCL:
   IF "AlwaysTRUE" THEN "Convert_analogs"(); END_IF;
END_REGION

REGION Network 45: Obsługa alarów
   RUNG wire#powerrail
      I_Contact( "FirstScan" )
      "Obsługa alarmów"()
   END_RUNG
   // the same network as SCL:
   IF NOT "FirstScan" THEN "Obsługa alarmów"(); END_IF;
END_REGION

REGION Network 46: Obsługa błędu Modbus TCP
   RUNG wire#powerrail
      I_Contact( "FirstScan" )
      "Błąd_Modbus_TCP"()
   END_RUNG
   // the same network as SCL:
   IF NOT "FirstScan" THEN "Błąd_Modbus_TCP"(); END_IF;
END_REGION

REGION Network 47: Inicjacja wartości startowych
   RUNG wire#powerrail
      I_Contact( "FirstScan" )
      Contact( "My_1Hz" )
      Contact( "IEC_Timer_Reset_delay_DB".Q )
      "dbSetup Write Parameters_KDN"()
   END_RUNG
   // the same network as SCL:
   IF NOT "FirstScan" AND "My_1Hz" AND "IEC_Timer_Reset_delay_DB".Q THEN
       "dbSetup Write Parameters_KDN"();   // "Inicjacja wartości startowych"
   END_IF;
END_REGION

REGION Network 48: Konversja Zmiennych
   RUNG wire#powerrail
      I_Contact( "FirstScan" )
      Contact( "IEC_Timer_Reset_delay_DB".Q )
      "Zmienne_SCADA"()
   END_RUNG
   // the same network as SCL:
   IF NOT "FirstScan" AND "IEC_Timer_Reset_delay_DB".Q THEN "Zmienne_SCADA"(); END_IF;
END_REGION

REGION Network 49: Konwersja zmiennej DLT czas na wartość liczbową
   RUNG wire#powerrail
      I_Contact( "FirstScan" )
      "Konwersja_Time_to_Int"()
   END_RUNG
   // the same network as SCL:
   IF NOT "FirstScan" THEN "Konwersja_Time_to_Int"(); END_IF;
END_REGION

REGION Network 50: Kontrola modelu sterowania pompownią
   RUNG wire#powerrail
      I_Contact( "FirstScan" )
      Contact( "IEC_Timer_Reset_delay_DB".Q )
      "Kontrola trybu sterowania"(Timer_Reset_delay := "IEC_Timer_Reset_delay_DB")
   END_RUNG
   // the same network as SCL:
   IF NOT "FirstScan" AND "IEC_Timer_Reset_delay_DB".Q THEN
       "Kontrola trybu sterowania"(Timer_Reset_delay := "IEC_Timer_Reset_delay_DB");
   END_IF;
END_REGION

REGION Network 51: Kontrola przyrostu ciśnienia
   // Funkcja w interwale czsowy sprawdza czy następuje przyrost czy spadekciśnienia
   // Wynik podawany jest do funkcji s"Sterowania dodatkową pompą" (Funkacja sterująca doączeniem pompy  dodatkowej)
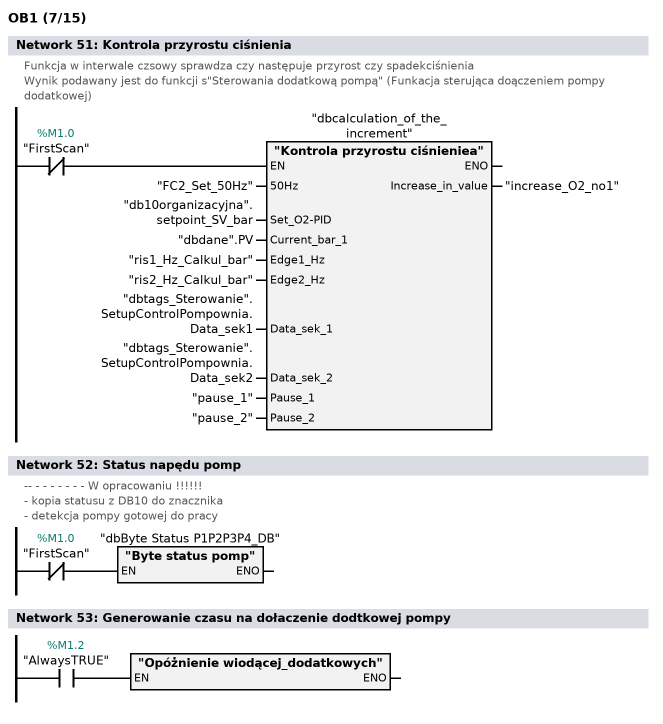
   RUNG wire#powerrail
      I_Contact( "FirstScan" )
      "dbcalculation_of_the_increment"("50Hz" := "FC2_Set_50Hz", "Set_O2-PID" := "db10organizacyjna".setpoint_SV_bar, Current_bar_1 := "dbdane".PV, Edge1_Hz := "ris1_Hz_Calkul_bar", Edge2_Hz := "ris2_Hz_Calkul_bar", Data_sek_1 := "dbtags_Sterowanie".SetupControlPompownia.Data_sek1, Data_sek_2 := "dbtags_Sterowanie".SetupControlPompownia.Data_sek2, Pause_1 := "pause_1", Pause_2 := "pause_2", Increase_in_value => "increase_O2_no1")
   END_RUNG
   // the same network as SCL:
   IF NOT "FirstScan" THEN
       "dbcalculation_of_the_increment"("50Hz" := "FC2_Set_50Hz",   // "Kontrola przyrostu ciśnieniea"
                               "Set_O2-PID" := "db10organizacyjna".setpoint_SV_bar,
                               Current_bar_1 := "dbdane".PV,
                               Edge1_Hz := "ris1_Hz_Calkul_bar",
                               Edge2_Hz := "ris2_Hz_Calkul_bar",
                               Data_sek_1 := "dbtags_Sterowanie".SetupControlPompownia.Data_sek1,
                               Data_sek_2 := "dbtags_Sterowanie".SetupControlPompownia.Data_sek2,
                               Pause_1 := "pause_1",
                               Pause_2 := "pause_2",
                               Increase_in_value => "increase_O2_no1");
   END_IF;
END_REGION

REGION Network 52: Status napędu pomp
   // -- - - - - - - - W opracowaniu !!!!!! 
   // - kopia statusu z DB10 do znacznika
   // - detekcja pompy gotowej do pracy
   RUNG wire#powerrail
      I_Contact( "FirstScan" )
      "dbByte Status P1P2P3P4_DB"()
   END_RUNG
   // the same network as SCL:
   IF NOT "FirstScan" THEN
       "dbByte Status P1P2P3P4_DB"();   // "Byte status pomp"
   END_IF;
END_REGION

REGION Network 53: Generowanie czasu na dołaczenie dodtkowej pompy
   RUNG wire#powerrail
      Contact( "AlwaysTRUE" )
      "Opóżnienie wiodącej_dodatkowych"()
   END_RUNG
   // the same network as SCL:
   IF "AlwaysTRUE" THEN "Opóżnienie wiodącej_dodatkowych"(); END_IF;
END_REGION

REGION Network 54: Sterowanie dołączeniem dodatkowych pomp
   // "dbdane".OUT_PURE_Real
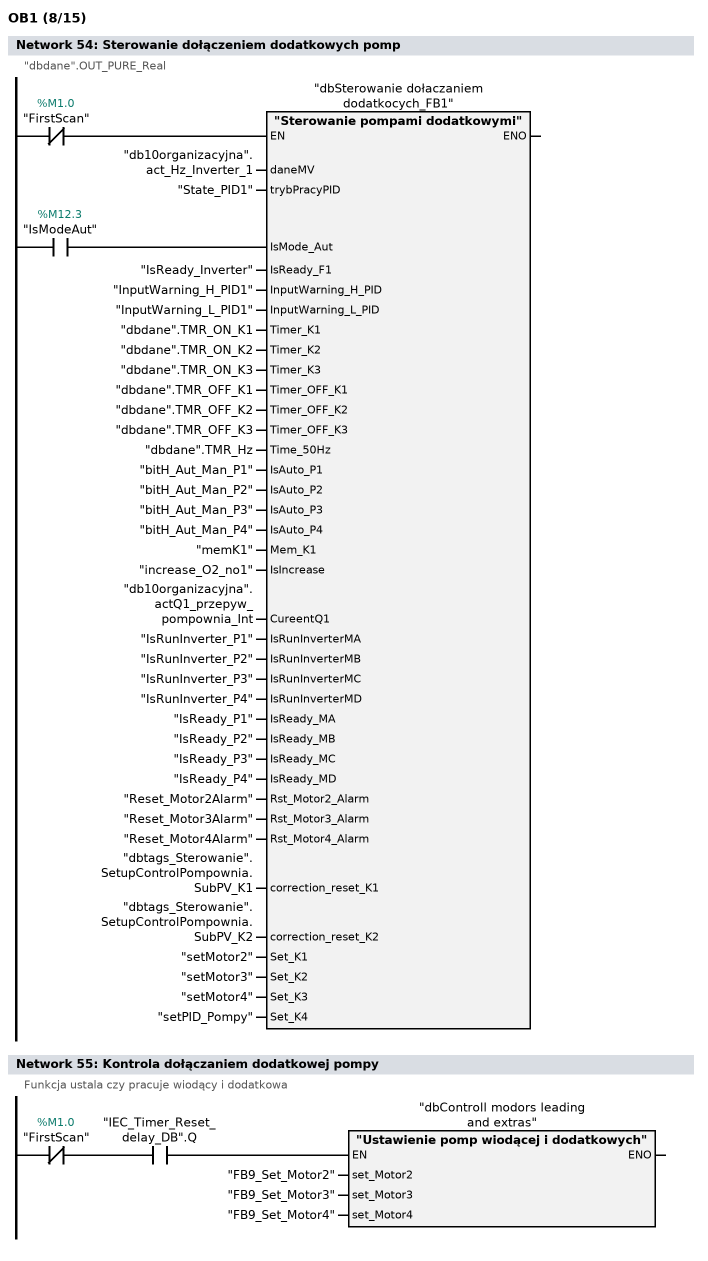
   RUNG wire#powerrail
      I_Contact( "FirstScan" )
      "dbSterowanie dołaczaniem dodatkocych_FB1"(IsMode_Aut := wire#w1, daneMV := "db10organizacyjna".act_Hz_Inverter_1, trybPracyPID := "State_PID1", IsReady_F1 := "IsReady_Inverter", InputWarning_H_PID := "InputWarning_H_PID1", InputWarning_L_PID := "InputWarning_L_PID1", Timer_K1 := "dbdane".TMR_ON_K1, Timer_K2 := "dbdane".TMR_ON_K2, Timer_K3 := "dbdane".TMR_ON_K3, Timer_OFF_K1 := "dbdane".TMR_OFF_K1, Timer_OFF_K2 := "dbdane".TMR_OFF_K2, Timer_OFF_K3 := "dbdane".TMR_OFF_K3, Time_50Hz := "dbdane".TMR_Hz, IsAuto_P1 := "bitH_Aut_Man_P1", IsAuto_P2 := "bitH_Aut_Man_P2", IsAuto_P3 := "bitH_Aut_Man_P3", IsAuto_P4 := "bitH_Aut_Man_P4", Mem_K1 := "memK1", IsIncrease := "increase_O2_no1", CureentQ1 := "db10organizacyjna".actQ1_przepyw_pompownia_Int, IsRunInverterMA := "IsRunInverter_P1", IsRunInverterMB := "IsRunInverter_P2", IsRunInverterMC := "IsRunInverter_P3", IsRunInverterMD := "IsRunInverter_P4", IsReady_MA := "IsReady_P1", IsReady_MB := "IsReady_P2", IsReady_MC := "IsReady_P3", IsReady_MD := "IsReady_P4", Rst_Motor2_Alarm := "Reset_Motor2Alarm", Rst_Motor3_Alarm := "Reset_Motor3Alarm", Rst_Motor4_Alarm := "Reset_Motor4Alarm", correction_reset_K1 := "dbtags_Sterowanie".SetupControlPompownia.SubPV_K1, correction_reset_K2 := "dbtags_Sterowanie".SetupControlPompownia.SubPV_K2, Set_K1 := "setMotor2", Set_K2 := "setMotor3", Set_K3 := "setMotor4", Set_K4 := "setPID_Pompy")
   END_RUNG
   RUNG wire#powerrail
      Contact( "IsModeAut" )
   END_RUNG wire#w1
   // the same network as SCL:
   IF NOT "FirstScan" THEN
       "dbSterowanie dołaczaniem dodatkocych_FB1"(daneMV := "db10organizacyjna".act_Hz_Inverter_1,   // "Sterowanie pompami dodatkowymi"
                               trybPracyPID := "State_PID1",
                               IsMode_Aut := "IsModeAut",
                               IsReady_F1 := "IsReady_Inverter",
                               InputWarning_H_PID := "InputWarning_H_PID1",
                               InputWarning_L_PID := "InputWarning_L_PID1",
                               Timer_K1 := "dbdane".TMR_ON_K1,
                               Timer_K2 := "dbdane".TMR_ON_K2,
                               Timer_K3 := "dbdane".TMR_ON_K3,
                               Timer_OFF_K1 := "dbdane".TMR_OFF_K1,
                               Timer_OFF_K2 := "dbdane".TMR_OFF_K2,
                               Timer_OFF_K3 := "dbdane".TMR_OFF_K3,
                               Time_50Hz := "dbdane".TMR_Hz,
                               IsAuto_P1 := "bitH_Aut_Man_P1",
                               IsAuto_P2 := "bitH_Aut_Man_P2",
                               IsAuto_P3 := "bitH_Aut_Man_P3",
                               IsAuto_P4 := "bitH_Aut_Man_P4",
                               Mem_K1 := "memK1",
                               IsIncrease := "increase_O2_no1",
                               CureentQ1 := "db10organizacyjna".actQ1_przepyw_pompownia_Int,
                               IsRunInverterMA := "IsRunInverter_P1",
                               IsRunInverterMB := "IsRunInverter_P2",
                               IsRunInverterMC := "IsRunInverter_P3",
                               IsRunInverterMD := "IsRunInverter_P4",
                               IsReady_MA := "IsReady_P1",
                               IsReady_MB := "IsReady_P2",
                               IsReady_MC := "IsReady_P3",
                               IsReady_MD := "IsReady_P4",
                               Rst_Motor2_Alarm := "Reset_Motor2Alarm",
                               Rst_Motor3_Alarm := "Reset_Motor3Alarm",
                               Rst_Motor4_Alarm := "Reset_Motor4Alarm",
                               correction_reset_K1 := "dbtags_Sterowanie".SetupControlPompownia.SubPV_K1,
                               correction_reset_K2 := "dbtags_Sterowanie".SetupControlPompownia.SubPV_K2,
                               Set_K1 := "setMotor2",
                               Set_K2 := "setMotor3",
                               Set_K3 := "setMotor4",
                               Set_K4 := "setPID_Pompy");
   END_IF;
END_REGION

REGION Network 55: Kontrola dołączaniem dodatkowej pompy
   // Funkcja ustala czy pracuje wiodący i dodatkowa
   RUNG wire#powerrail
      I_Contact( "FirstScan" )
      Contact( "IEC_Timer_Reset_delay_DB".Q )
      "dbControll modors leading and extras"(set_Motor2 := "FB9_Set_Motor2", set_Motor3 := "FB9_Set_Motor3", set_Motor4 := "FB9_Set_Motor4")
   END_RUNG
   // the same network as SCL:
   IF NOT "FirstScan" AND "IEC_Timer_Reset_delay_DB".Q THEN
       "dbControll modors leading and extras"(set_Motor2 := "FB9_Set_Motor2",   // "Ustawienie pomp wiodącej i dodatkowych"
                               set_Motor3 := "FB9_Set_Motor3",
                               set_Motor4 := "FB9_Set_Motor4");
   END_IF;
END_REGION

REGION Network 56: Falownik P1
   // Sterowaniem pracy z falownika. Sterowanie napędem na pozycji MC
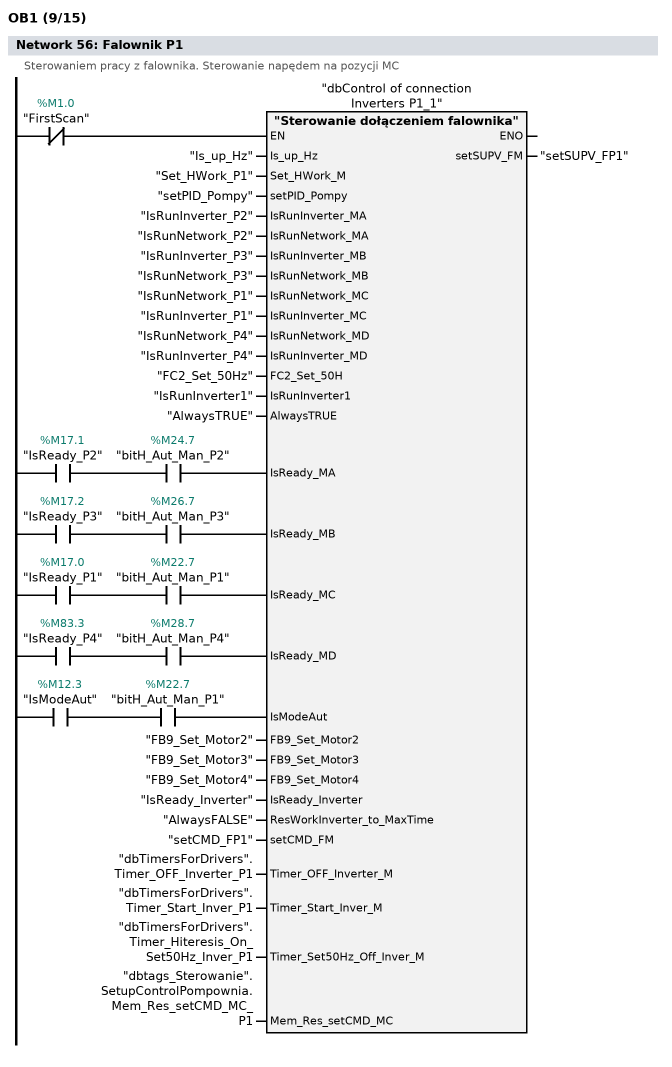
   RUNG wire#powerrail
      I_Contact( "FirstScan" )
      "dbControl of connection Inverters P1_1"(IsReady_MA := wire#w1, IsReady_MB := wire#w2, IsReady_MC := wire#w3, IsReady_MD := wire#w4, IsModeAut := wire#w5, Is_up_Hz := "Is_up_Hz", Set_HWork_M := "Set_HWork_P1", setPID_Pompy := "setPID_Pompy", IsRunInverter_MA := "IsRunInverter_P2", IsRunNetwork_MA := "IsRunNetwork_P2", IsRunInverter_MB := "IsRunInverter_P3", IsRunNetwork_MB := "IsRunNetwork_P3", IsRunNetwork_MC := "IsRunNetwork_P1", IsRunInverter_MC := "IsRunInverter_P1", IsRunNetwork_MD := "IsRunNetwork_P4", IsRunInverter_MD := "IsRunInverter_P4", FC2_Set_50H := "FC2_Set_50Hz", IsRunInverter1 := "IsRunInverter1", AlwaysTRUE := "AlwaysTRUE", FB9_Set_Motor2 := "FB9_Set_Motor2", FB9_Set_Motor3 := "FB9_Set_Motor3", FB9_Set_Motor4 := "FB9_Set_Motor4", IsReady_Inverter := "IsReady_Inverter", ResWorkInverter_to_MaxTime := "AlwaysFALSE", setCMD_FM := "setCMD_FP1", Timer_OFF_Inverter_M := "dbTimersForDrivers".Timer_OFF_Inverter_P1, Timer_Start_Inver_M := "dbTimersForDrivers".Timer_Start_Inver_P1, Timer_Set50Hz_Off_Inver_M := "dbTimersForDrivers".Timer_Hiteresis_On_Set50Hz_Inver_P1, Mem_Res_setCMD_MC := "dbtags_Sterowanie".SetupControlPompownia.Mem_Res_setCMD_MC_P1, setSUPV_FM => "setSUPV_FP1")
   END_RUNG
   RUNG wire#powerrail
      Contact( "IsReady_P2" )
      Contact( "bitH_Aut_Man_P2" )
   END_RUNG wire#w1
   RUNG wire#powerrail
      Contact( "IsReady_P3" )
      Contact( "bitH_Aut_Man_P3" )
   END_RUNG wire#w2
   RUNG wire#powerrail
      Contact( "IsReady_P1" )
      Contact( "bitH_Aut_Man_P1" )
   END_RUNG wire#w3
   RUNG wire#powerrail
      Contact( "IsReady_P4" )
      Contact( "bitH_Aut_Man_P4" )
   END_RUNG wire#w4
   RUNG wire#powerrail
      Contact( "IsModeAut" )
      Contact( "bitH_Aut_Man_P1" )
   END_RUNG wire#w5
   // the same network as SCL:
   IF NOT "FirstScan" THEN
       "dbControl of connection Inverters P1_1"(Is_up_Hz := "Is_up_Hz",   // "Sterowanie dołączeniem falownika"
                               Set_HWork_M := "Set_HWork_P1",
                               setPID_Pompy := "setPID_Pompy",
                               IsRunInverter_MA := "IsRunInverter_P2",
                               IsRunNetwork_MA := "IsRunNetwork_P2",
                               IsRunInverter_MB := "IsRunInverter_P3",
                               IsRunNetwork_MB := "IsRunNetwork_P3",
                               IsRunNetwork_MC := "IsRunNetwork_P1",
                               IsRunInverter_MC := "IsRunInverter_P1",
                               IsRunNetwork_MD := "IsRunNetwork_P4",
                               IsRunInverter_MD := "IsRunInverter_P4",
                               FC2_Set_50H := "FC2_Set_50Hz",
                               IsRunInverter1 := "IsRunInverter1",
                               AlwaysTRUE := "AlwaysTRUE",
                               IsReady_MA := "IsReady_P2" AND "bitH_Aut_Man_P2",
                               IsReady_MB := "IsReady_P3" AND "bitH_Aut_Man_P3",
                               IsReady_MC := "IsReady_P1" AND "bitH_Aut_Man_P1",
                               IsReady_MD := "IsReady_P4" AND "bitH_Aut_Man_P4",
                               IsModeAut := "IsModeAut" AND "bitH_Aut_Man_P1",
                               FB9_Set_Motor2 := "FB9_Set_Motor2",
                               FB9_Set_Motor3 := "FB9_Set_Motor3",
                               FB9_Set_Motor4 := "FB9_Set_Motor4",
                               IsReady_Inverter := "IsReady_Inverter",
                               ResWorkInverter_to_MaxTime := "AlwaysFALSE",
                               setCMD_FM := "setCMD_FP1",
                               Timer_OFF_Inverter_M := "dbTimersForDrivers".Timer_OFF_Inverter_P1,
                               Timer_Start_Inver_M := "dbTimersForDrivers".Timer_Start_Inver_P1,
                               Timer_Set50Hz_Off_Inver_M := "dbTimersForDrivers".Timer_Hiteresis_On_Set50Hz_Inver_P1,
                               Mem_Res_setCMD_MC := "dbtags_Sterowanie".SetupControlPompownia.Mem_Res_setCMD_MC_P1,
                               setSUPV_FM => "setSUPV_FP1");
   END_IF;
END_REGION

REGION Network 57: Falownik P2
   // Sterowaniem pracy z falownika. Sterowanie napędem na pozycji MC
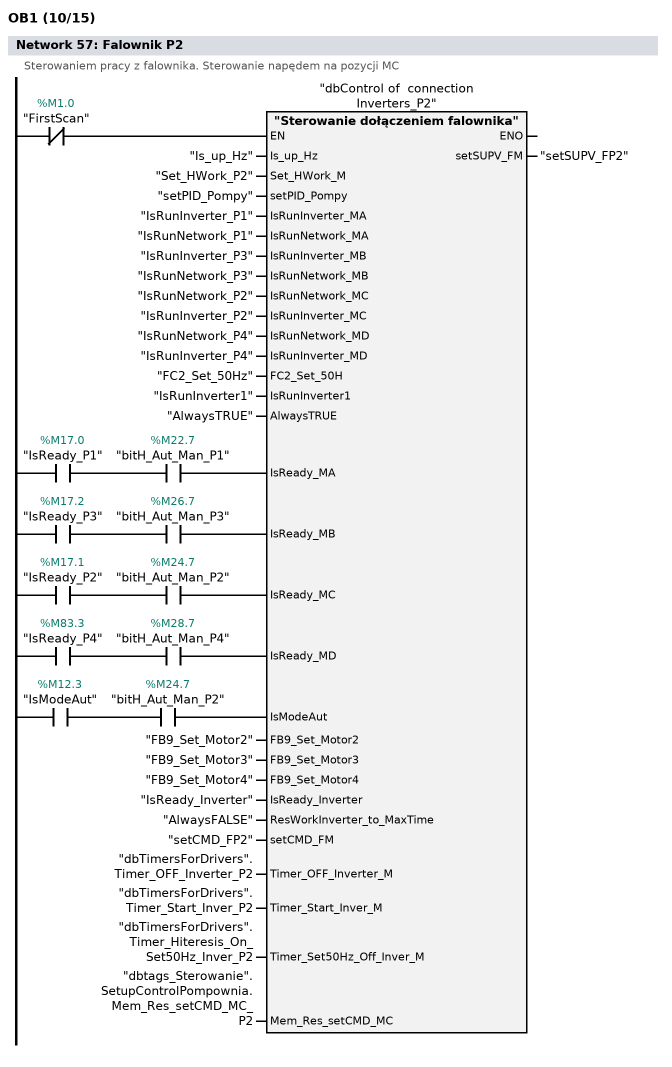
   RUNG wire#powerrail
      I_Contact( "FirstScan" )
      "dbControl of  connection Inverters_P2"(IsReady_MA := wire#w1, IsReady_MB := wire#w2, IsReady_MC := wire#w3, IsReady_MD := wire#w4, IsModeAut := wire#w5, Is_up_Hz := "Is_up_Hz", Set_HWork_M := "Set_HWork_P2", setPID_Pompy := "setPID_Pompy", IsRunInverter_MA := "IsRunInverter_P1", IsRunNetwork_MA := "IsRunNetwork_P1", IsRunInverter_MB := "IsRunInverter_P3", IsRunNetwork_MB := "IsRunNetwork_P3", IsRunNetwork_MC := "IsRunNetwork_P2", IsRunInverter_MC := "IsRunInverter_P2", IsRunNetwork_MD := "IsRunNetwork_P4", IsRunInverter_MD := "IsRunInverter_P4", FC2_Set_50H := "FC2_Set_50Hz", IsRunInverter1 := "IsRunInverter1", AlwaysTRUE := "AlwaysTRUE", FB9_Set_Motor2 := "FB9_Set_Motor2", FB9_Set_Motor3 := "FB9_Set_Motor3", FB9_Set_Motor4 := "FB9_Set_Motor4", IsReady_Inverter := "IsReady_Inverter", ResWorkInverter_to_MaxTime := "AlwaysFALSE", setCMD_FM := "setCMD_FP2", Timer_OFF_Inverter_M := "dbTimersForDrivers".Timer_OFF_Inverter_P2, Timer_Start_Inver_M := "dbTimersForDrivers".Timer_Start_Inver_P2, Timer_Set50Hz_Off_Inver_M := "dbTimersForDrivers".Timer_Hiteresis_On_Set50Hz_Inver_P2, Mem_Res_setCMD_MC := "dbtags_Sterowanie".SetupControlPompownia.Mem_Res_setCMD_MC_P2, setSUPV_FM => "setSUPV_FP2")
   END_RUNG
   RUNG wire#powerrail
      Contact( "IsReady_P1" )
      Contact( "bitH_Aut_Man_P1" )
   END_RUNG wire#w1
   RUNG wire#powerrail
      Contact( "IsReady_P3" )
      Contact( "bitH_Aut_Man_P3" )
   END_RUNG wire#w2
   RUNG wire#powerrail
      Contact( "IsReady_P2" )
      Contact( "bitH_Aut_Man_P2" )
   END_RUNG wire#w3
   RUNG wire#powerrail
      Contact( "IsReady_P4" )
      Contact( "bitH_Aut_Man_P4" )
   END_RUNG wire#w4
   RUNG wire#powerrail
      Contact( "IsModeAut" )
      Contact( "bitH_Aut_Man_P2" )
   END_RUNG wire#w5
   // the same network as SCL:
   IF NOT "FirstScan" THEN
       "dbControl of  connection Inverters_P2"(Is_up_Hz := "Is_up_Hz",   // "Sterowanie dołączeniem falownika"
                               Set_HWork_M := "Set_HWork_P2",
                               setPID_Pompy := "setPID_Pompy",
                               IsRunInverter_MA := "IsRunInverter_P1",
                               IsRunNetwork_MA := "IsRunNetwork_P1",
                               IsRunInverter_MB := "IsRunInverter_P3",
                               IsRunNetwork_MB := "IsRunNetwork_P3",
                               IsRunNetwork_MC := "IsRunNetwork_P2",
                               IsRunInverter_MC := "IsRunInverter_P2",
                               IsRunNetwork_MD := "IsRunNetwork_P4",
                               IsRunInverter_MD := "IsRunInverter_P4",
                               FC2_Set_50H := "FC2_Set_50Hz",
                               IsRunInverter1 := "IsRunInverter1",
                               AlwaysTRUE := "AlwaysTRUE",
                               IsReady_MA := "IsReady_P1" AND "bitH_Aut_Man_P1",
                               IsReady_MB := "IsReady_P3" AND "bitH_Aut_Man_P3",
                               IsReady_MC := "IsReady_P2" AND "bitH_Aut_Man_P2",
                               IsReady_MD := "IsReady_P4" AND "bitH_Aut_Man_P4",
                               IsModeAut := "IsModeAut" AND "bitH_Aut_Man_P2",
                               FB9_Set_Motor2 := "FB9_Set_Motor2",
                               FB9_Set_Motor3 := "FB9_Set_Motor3",
                               FB9_Set_Motor4 := "FB9_Set_Motor4",
                               IsReady_Inverter := "IsReady_Inverter",
                               ResWorkInverter_to_MaxTime := "AlwaysFALSE",
                               setCMD_FM := "setCMD_FP2",
                               Timer_OFF_Inverter_M := "dbTimersForDrivers".Timer_OFF_Inverter_P2,
                               Timer_Start_Inver_M := "dbTimersForDrivers".Timer_Start_Inver_P2,
                               Timer_Set50Hz_Off_Inver_M := "dbTimersForDrivers".Timer_Hiteresis_On_Set50Hz_Inver_P2,
                               Mem_Res_setCMD_MC := "dbtags_Sterowanie".SetupControlPompownia.Mem_Res_setCMD_MC_P2,
                               setSUPV_FM => "setSUPV_FP2");
   END_IF;
END_REGION

